KUKA KRL program: MyProgram_100().src

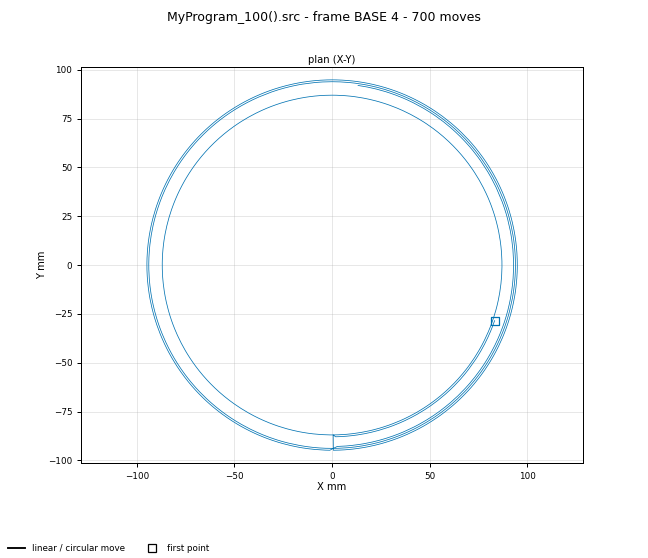
[picture p0: tool path of MyProgram_100().src in frame BASE 4, 700 of 700 moves have a stored position in this frame; points joined in program order, loops and branches not executed]
&ACCESS RVP
&REL 1
&PARAM TEMPLATE = C:\KRC\Roboter\Template\vorgabe
&PARAM EDITMASK = *
DEF MyProgram_100()
; ---- Setting reference (Base) ----
$BASE = BASE_DATA[4]

; --------------------------
; ---- Setting tool (TCP) ----
$TOOL = TOOL_DATA[3]
; --------------------------

$VEL.CP = VEL_APROX_PRINT
Startdeposition()
$VEL.CP = VEL_PRINT
LIN {X 83.2167,Y -28.4567,Z 91,A -24.2828,B 24.9207,C -2.0559,E1 25.1508,E2 469.2806} C_DIS
LIN {X 82.0556,Y -31.6498,Z 91,A -26.2319,B 24.9206,C -2.0583,E1 25.1489,E2 471.2131} C_DIS
LIN {X 81.1855,Y -33.8182,Z 91,A -28.5047,B 24.9229,C -2.0275,E1 25.1464,E2 473.5461} C_DIS
LIN {X 79.8483,Y -36.8641,Z 91,A -30.8218,B 24.9238,C -2.0158,E1 25.1436,E2 475.8782} C_DIS
LIN {X 78.1167,Y -40.407,Z 91,A -33.4521,B 24.9245,C -2.0061,E1 25.1403,E2 478.5174} C_DIS
LIN {X 76.1397,Y -44.0179,Z 91,A -35.2877,B 24.9229,C -2.0276,E1 25.1378,E2 480.2928} C_DIS
LIN {X 74.5815,Y -46.6088,Z 91,A -36.9718,B 24.9226,C -2.032,E1 25.1354,E2 481.958} C_DIS
LIN {X 73.464,Y -48.3511,Z 91,A -38.6448,B 24.9237,C -2.0169,E1 25.1328,E2 483.6583} C_DIS
LIN {X 69.7273,Y -53.5994,Z 91,A -42.6293,B 24.924,C -2.0128,E1 25.1263,E2 487.6331} C_DIS
LIN {X 67.7377,Y -56.0928,Z 91,A -44.8775,B 24.9249,C -2.0014,E1 25.1223,E2 489.8977} C_DIS
LIN {X 65.6016,Y -58.5766,Z 91,A -47.8573,B 24.9275,C -1.967,E1 25.1167,E2 492.9454} C_DIS
LIN {X 62.5852,Y -61.7889,Z 91,A -49.8249,B 24.9257,C -1.9908,E1 25.113,E2 494.8484} C_DIS
LIN {X 60.3828,Y -63.9431,Z 91,A -51.8518,B 24.9261,C -1.9854,E1 25.1089,E2 496.8799} C_DIS
LIN {X 57.9684,Y -66.1397,Z 91,A -54.9821,B 24.929,C -1.9464,E1 25.1022,E2 500.0897} C_DIS
LIN {X 54.1399,Y -69.31,Z 91,A -57.5673,B 24.9279,C -1.9614,E1 25.0966,E2 502.63} C_DIS
LIN {X 50.5294,Y -71.9838,Z 91,A -60.0241,B 24.9271,C -1.9713,E1 25.0911,E2 505.0547} C_DIS
LIN {X 47.6024,Y -73.9513,Z 91,A -62.3164,B 24.9275,C -1.967,E1 25.0858,E2 507.3495} C_DIS
LIN {X 43.6058,Y -76.3765,Z 91,A -65.9359,B 24.9293,C -1.9421,E1 25.0769,E2 511.0167} C_DIS
LIN {X 40.7609,Y -77.9317,Z 91,A -67.6031,B 24.9285,C -1.9534,E1 25.0729,E2 512.6526} C_DIS
LIN {X 37.3321,Y -79.6313,Z 91,A -69.9938,B 24.9285,C -1.9529,E1 25.0669,E2 515.0382} C_DIS
LIN {X 34.5175,Y -80.891,Z 91,A -72.0438,B 24.9288,C -1.9485,E1 25.0617,E2 517.0937} C_DIS
LIN {X 31.395,Y -82.1533,Z 91,A -73.9789,B 24.9284,C -1.9541,E1 25.0567,E2 519.0112} C_DIS
LIN {X 29.0169,Y -83.0229,Z 91,A -76.1026,B 24.9297,C -1.9362,E1 25.051,E2 521.1729} C_DIS
LIN {X 23.7913,Y -84.6686,Z 91,A -79.5291,B 24.9297,C -1.9368,E1 25.0419,E2 524.5919} C_DIS
LIN {X 20.0098,Y -85.6413,Z 91,A -82.0028,B 24.9297,C -1.9366,E1 25.0352,E2 527.0625} C_DIS
LIN {X 16.5913,Y -86.3684,Z 91,A -84.3026,B 24.9299,C -1.9339,E1 25.0288,E2 529.3658} C_DIS
LIN {X 13.0968,Y -86.9676,Z 91,A -86.358,B 24.9294,C -1.9405,E1 25.0232,E2 531.4036} C_DIS
LIN {X 10.7294,Y -87.291,Z 91,A -88.0802,B 24.9299,C -1.9341,E1 25.0184,E2 533.1395} C_DIS
LIN {X 7.6095,Y -87.6177,Z 91,A -90.1493,B 24.93,C -1.9322,E1 25.0127,E2 535.2119} C_DIS
LIN {X 4.3054,Y -87.8424,Z 91,A -92.3321,B 24.9301,C -1.9305,E1 25.0066,E2 537.3979} C_DIS
LIN {X 1.8163,Y -87.929,Z 91,A -93.8282,B 24.9299,C -1.934,E1 25.0024,E2 538.8854} C_DIS
LIN {X 1.8163,Y -87.929,Z 91,A -93.8282,B 24.9299,C -1.934,E1 25.0024,E2 538.8854} C_DIS
Enddeposition()
LIN {X 0.5508,Y -86.9757,Z 91,A -94.1889,B 24.9276,C -1.9656,E1 25.0016,E2 539.171} C_DIS
Startdeposition()
$VEL.CP = VEL_PRINT
LIN {X 3.2037,Y -86.9212,Z 91,A -92.2114,B 24.927,C -1.9735,E1 25.0072,E2 537.1751} C_DIS
LIN {X 5.3312,Y -86.8173,Z 91,A -90.8306,B 24.927,C -1.9734,E1 25.011,E2 535.7952} C_DIS
LIN {X 7.5293,Y -86.6532,Z 91,A -89.1451,B 24.9264,C -1.9817,E1 25.0158,E2 534.0908} C_DIS
LIN {X 10.6333,Y -86.3277,Z 91,A -87.3159,B 24.9268,C -1.9755,E1 25.0208,E2 532.2777} C_DIS
LIN {X 12.6686,Y -86.0529,Z 91,A -85.9635,B 24.9268,C -1.9764,E1 25.0246,E2 530.9243} C_DIS
LIN {X 14.7955,Y -85.7133,Z 91,A -84.5308,B 24.9266,C -1.9779,E1 25.0285,E2 529.4895} C_DIS
LIN {X 16.8911,Y -85.3246,Z 91,A -83.0893,B 24.9265,C -1.9803,E1 25.0325,E2 528.0439} C_DIS
LIN {X 19.0492,Y -84.8684,Z 91,A -81.6996,B 24.9265,C -1.9796,E1 25.0363,E2 526.6578} C_DIS
LIN {X 21.1564,Y -84.3677,Z 91,A -80.0242,B 24.9258,C -1.9892,E1 25.0409,E2 524.9621} C_DIS
LIN {X 24.1141,Y -83.57,Z 91,A -78.2555,B 24.9263,C -1.9832,E1 25.0456,E2 523.2107} C_DIS
LIN {X 26.0935,Y -82.9736,Z 91,A -76.8469,B 24.926,C -1.9863,E1 25.0493,E2 521.7972} C_DIS
LIN {X 28.8765,Y -82.0464,Z 91,A -74.8223,B 24.9256,C -1.9918,E1 25.0547,E2 519.7636} C_DIS
LIN {X 31.1689,Y -81.2034,Z 91,A -73.2999,B 24.9256,C -1.9911,E1 25.0587,E2 518.2461} C_DIS
LIN {X 33.2121,Y -80.389,Z 91,A -71.9115,B 24.9256,C -1.9911,E1 25.0623,E2 516.8608} C_DIS
LIN {X 35.1707,Y -79.5517,Z 91,A -70.5232,B 24.9256,C -1.9927,E1 25.0658,E2 515.472} C_DIS
LIN {X 37.1076,Y -78.6671,Z 91,A -68.9087,B 24.9248,C -2.002,E1 25.0699,E2 513.8396} C_DIS
LIN {X 39.9862,Y -77.2445,Z 91,A -66.7842,B 24.9246,C -2.0058,E1 25.0752,E2 511.712} C_DIS
LIN {X 42.7562,Y -75.7465,Z 91,A -64.9422,B 24.9249,C -2.0016,E1 25.0797,E2 509.8854} C_DIS
LIN {X 44.5558,Y -74.7018,Z 91,A -63.5773,B 24.9247,C -2.0039,E1 25.083,E2 508.5192} C_DIS
LIN {X 47.0289,Y -73.1693,Z 91,A -61.5921,B 24.9243,C -2.0099,E1 25.0877,E2 506.5262} C_DIS
LIN {X 48.8455,Y -71.9694,Z 91,A -60.1397,B 24.924,C -2.0133,E1 25.0911,E2 505.0705} C_DIS
LIN {X 50.8905,Y -70.539,Z 91,A -58.5953,B 24.924,C -2.0133,E1 25.0946,E2 503.5315} C_DIS
LIN {X 53.0933,Y -68.8953,Z 91,A -56.6917,B 24.9235,C -2.0203,E1 25.0988,E2 501.6182} C_DIS
LIN {X 55.5445,Y -66.9349,Z 91,A -54.6246,B 24.9231,C -2.0248,E1 25.1033,E2 499.5482} C_DIS
LIN {X 57.9872,Y -64.8302,Z 91,A -52.4847,B 24.9227,C -2.0302,E1 25.1078,E2 497.4041} C_DIS
LIN {X 60.3294,Y -62.6564,Z 91,A -50.4216,B 24.9224,C -2.0338,E1 25.112,E2 495.3411} C_DIS
LIN {X 62.6022,Y -60.3857,Z 91,A -48.3282,B 24.9221,C -2.0382,E1 25.1161,E2 493.2463} C_DIS
LIN {X 64.7171,Y -58.1135,Z 91,A -46.2361,B 24.9216,C -2.0449,E1 25.1201,E2 491.1474} C_DIS
LIN {X 66.8928,Y -55.5951,Z 91,A -44.092,B 24.9213,C -2.0489,E1 25.1239,E2 489.0036} C_DIS
LIN {X 68.8721,Y -53.1234,Z 91,A -42.0124,B 24.9209,C -2.0543,E1 25.1275,E2 486.9213} C_DIS
LIN {X 70.4344,Y -51.0353,Z 91,A -40.4263,B 24.9209,C -2.0543,E1 25.1301,E2 485.3426} C_DIS
LIN {X 71.6523,Y -49.311,Z 91,A -39.0478,B 24.9206,C -2.0578,E1 25.1323,E2 483.9628} C_DIS
LIN {X 72.9068,Y -47.4363,Z 91,A -37.6066,B 24.9204,C -2.0604,E1 25.1346,E2 482.5226} C_DIS
LIN {X 74.0526,Y -45.6272,Z 91,A -36.1871,B 24.9201,C -2.0647,E1 25.1367,E2 481.1002} C_DIS
LIN {X 75.1471,Y -43.8021,Z 91,A -34.6258,B 24.9193,C -2.0743,E1 25.1389,E2 479.5242} C_DIS
LIN {X 76.6816,Y -41.0553,Z 91,A -32.7076,B 24.9193,C -2.0749,E1 25.1415,E2 477.6144} C_DIS
LIN {X 77.9149,Y -38.6618,Z 91,A -30.7952,B 24.9185,C -2.085,E1 25.1439,E2 475.6884} C_DIS
LIN {X 79.0625,Y -36.2567,Z 91,A -29.2221,B 24.9185,C -2.0839,E1 25.1457,E2 474.1264} C_DIS
LIN {X 79.915,Y -34.3382,Z 91,A -27.8263,B 24.9182,C -2.0885,E1 25.1473,E2 472.7273} C_DIS
LIN {X 81.0139,Y -31.6582,Z 91,A -25.823,B 24.9175,C -2.0977,E1 25.1494,E2 470.7135} C_DIS
LIN {X 81.8944,Y -29.306,Z 91,A -24.3434,B 24.9175,C -2.0967,E1 25.1508,E2 469.2445} C_DIS
LIN {X 82.564,Y -27.3612,Z 91,A -22.9651,B 24.9172,C -2.1017,E1 25.152,E2 467.8621} C_DIS
LIN {X 83.2312,Y -25.2607,Z 91,A -21.5144,B 24.9168,C -2.1062,E1 25.1532,E2 466.4091} C_DIS
LIN {X 83.8304,Y -23.1943,Z 91,A -20.1436,B 24.9166,C -2.109,E1 25.1543,E2 465.0394} C_DIS
LIN {X 84.4419,Y -20.8587,Z 91,A -18.3066,B 24.9155,C -2.1227,E1 25.1555,E2 463.1807} C_DIS
LIN {X 85.0643,Y -18.1527,Z 91,A -16.7409,B 24.9158,C -2.1193,E1 25.1565,E2 461.6323} C_DIS
LIN {X 85.4869,Y -16.0474,Z 91,A -15.3263,B 24.9154,C -2.1238,E1 25.1572,E2 460.2153} C_DIS
LIN {X 85.8311,Y -14.0906,Z 91,A -13.9881,B 24.915,C -2.129,E1 25.1579,E2 458.8727} C_DIS
LIN {X 86.1885,Y -11.7095,Z 91,A -12.4573,B 24.9147,C -2.1321,E1 25.1585,E2 457.3435} C_DIS
LIN {X 86.4429,Y -9.6511,Z 91,A -11.0636,B 24.9143,C -2.1375,E1 25.1589,E2 455.9454} C_DIS
LIN {X 86.653,Y -7.5314,Z 91,A -9.7473,B 24.9142,C -2.139,E1 25.1593,E2 454.6334} C_DIS
LIN {X 86.8123,Y -5.4068,Z 91,A -8.2791,B 24.9136,C -2.1457,E1 25.1595,E2 453.158} C_DIS
LIN {X 86.9211,Y -3.2052,Z 91,A -6.8454,B 24.9133,C -2.1497,E1 25.1597,E2 451.7233} C_DIS
LIN {X 86.9756,Y -0.9547,Z 91,A -5.1249,B 24.9123,C -2.1628,E1 25.1597,E2 449.9821} C_DIS
LIN {X 86.9553,Y 2.0675,Z 91,A -3.3966,B 24.9125,C -2.16,E1 25.1597,E2 448.2709} C_DIS
LIN {X 86.8784,Y 4.1974,Z 91,A -2.0346,B 24.9122,C -2.163,E1 25.1595,E2 446.9098} C_DIS
LIN {X 86.7456,Y 6.3985,Z 91,A -0.2652,B 24.911,C -2.1787,E1 25.1592,E2 445.1138} C_DIS
LIN {X 86.4587,Y 9.5085,Z 91,A 1.6567,B 24.9108,C -2.1805,E1 25.1586,E2 443.1991} C_DIS
LIN {X 86.0492,Y 12.6942,Z 91,A 3.568,B 24.9108,C -2.18,E1 25.1579,E2 441.3003} C_DIS
LIN {X 85.7127,Y 14.7989,Z 91,A 4.9825,B 24.9105,C -2.1847,E1 25.1573,E2 439.883} C_DIS
LIN {X 85.3239,Y 16.8945,Z 91,A 6.4155,B 24.91,C -2.1901,E1 25.1565,E2 438.4456} C_DIS
LIN {X 84.8193,Y 19.2669,Z 91,A 8.1959,B 24.9091,C -2.2014,E1 25.1554,E2 436.6488} C_DIS
LIN {X 84.1069,Y 22.1706,Z 91,A 9.9085,B 24.9093,C -2.1985,E1 25.1543,E2 434.9531} C_DIS
LIN {X 83.3271,Y 24.9422,Z 91,A 11.8642,B 24.9087,C -2.2062,E1 25.1527,E2 432.9902} C_DIS
LIN {X 82.624,Y 27.1791,Z 91,A 13.4914,B 24.9081,C -2.2137,E1 25.1513,E2 431.3545} C_DIS
LIN {X 81.5552,Y 30.2355,Z 91,A 15.4262,B 24.9081,C -2.2131,E1 25.1495,E2 429.432} C_DIS
LIN {X 80.8419,Y 32.0944,Z 91,A 16.802,B 24.9076,C -2.2192,E1 25.1481,E2 428.0496} C_DIS
LIN {X 79.9497,Y 34.2571,Z 91,A 18.2728,B 24.9075,C -2.2211,E1 25.1465,E2 426.5821} C_DIS
LIN {X 78.9634,Y 36.4723,Z 91,A 20.0777,B 24.9065,C -2.2329,E1 25.1444,E2 424.7595} C_DIS
LIN {X 77.4059,Y 39.6711,Z 91,A 22.3006,B 24.9063,C -2.2352,E1 25.1417,E2 422.5429} C_DIS
LIN {X 76.1964,Y 41.9495,Z 91,A 23.857,B 24.9063,C -2.2349,E1 25.1396,E2 420.9954} C_DIS
LIN {X 75.2363,Y 43.6472,Z 91,A 25.1847,B 24.9059,C -2.2398,E1 25.1378,E2 419.663} C_DIS
LIN {X 74.0934,Y 45.5609,Z 91,A 26.6123,B 24.9057,C -2.2422,E1 25.1357,E2 418.2368} C_DIS
LIN {X 72.9171,Y 47.4205,Z 91,A 28.0297,B 24.9055,C -2.2449,E1 25.1336,E2 416.8203} C_DIS
LIN {X 71.7788,Y 49.1265,Z 91,A 29.5574,B 24.9047,C -2.2544,E1 25.1311,E2 415.2777} C_DIS
LIN {X 69.8641,Y 51.8135,Z 91,A 31.5363,B 24.9047,C -2.2531,E1 25.1279,E2 413.3115} C_DIS
LIN {X 68.2433,Y 53.9289,Z 91,A 33.4574,B 24.9039,C -2.263,E1 25.1246,E2 411.3761} C_DIS
LIN {X 66.2325,Y 56.3801,Z 91,A 35.528,B 24.9036,C -2.2672,E1 25.1209,E2 409.3049} C_DIS
LIN {X 64.0975,Y 58.7961,Z 91,A 37.6276,B 24.9032,C -2.2712,E1 25.117,E2 407.2053} C_DIS
LIN {X 61.9023,Y 61.103,Z 91,A 39.6528,B 24.9031,C -2.2732,E1 25.113,E2 405.184} C_DIS
LIN {X 59.6715,Y 63.2834,Z 91,A 41.8334,B 24.9023,C -2.2817,E1 25.1086,E2 402.9923} C_DIS
LIN {X 56.806,Y 65.8694,Z 91,A 44.381,B 24.9019,C -2.2869,E1 25.1033,E2 400.4426} C_DIS
LIN {X 54.3557,Y 67.9053,Z 91,A 46.4557,B 24.9016,C -2.29,E1 25.0988,E2 398.3685} C_DIS
LIN {X 51.8327,Y 69.8498,Z 91,A 48.3364,B 24.9019,C -2.2865,E1 25.0946,E2 396.5029} C_DIS
LIN {X 50.1143,Y 71.0928,Z 91,A 49.7213,B 24.9017,C -2.2884,E1 25.0915,E2 395.1183} C_DIS
LIN {X 48.3276,Y 72.32,Z 91,A 51.2092,B 24.9014,C -2.2927,E1 25.088,E2 393.6251} C_DIS
LIN {X 46.6021,Y 73.443,Z 91,A 52.7575,B 24.9006,C -2.3012,E1 25.0844,E2 392.0617} C_DIS
LIN {X 43.7946,Y 75.1514,Z 91,A 54.6744,B 24.9011,C -2.2962,E1 25.0798,E2 390.1627} C_DIS
LIN {X 42.1288,Y 76.0968,Z 91,A 55.9691,B 24.9008,C -2.299,E1 25.0767,E2 388.865} C_DIS
LIN {X 40.1328,Y 77.1678,Z 91,A 57.3992,B 24.9008,C -2.299,E1 25.0731,E2 387.4391} C_DIS
LIN {X 38.2334,Y 78.1259,Z 91,A 58.8479,B 24.9006,C -2.3023,E1 25.0695,E2 385.9864} C_DIS
LIN {X 36.2219,Y 79.0785,Z 91,A 60.4307,B 24.9001,C -2.3078,E1 25.0655,E2 384.3945} C_DIS
LIN {X 33.3591,Y 80.328,Z 91,A 62.3607,B 24.9002,C -2.3059,E1 25.0605,E2 382.4738} C_DIS
LIN {X 31.3818,Y 81.1218,Z 91,A 63.6826,B 24.9004,C -2.3046,E1 25.0571,E2 381.1578} C_DIS
LIN {X 29.3004,Y 81.8964,Z 91,A 65.1628,B 24.9002,C -2.3065,E1 25.0532,E2 379.6762} C_DIS
LIN {X 26.8533,Y 82.7307,Z 91,A 67.0718,B 24.8995,C -2.3146,E1 25.0481,E2 377.7517} C_DIS
LIN {X 24.308,Y 83.5139,Z 91,A 68.6499,B 24.8999,C -2.3102,E1 25.0439,E2 376.1869} C_DIS
LIN {X 22.2486,Y 84.0865,Z 91,A 70.2341,B 24.8993,C -2.3167,E1 25.0396,E2 374.5896} C_DIS
LIN {X 19.099,Y 84.8571,Z 91,A 72.3825,B 24.8992,C -2.3183,E1 25.0338,E2 372.4406} C_DIS
LIN {X 15.918,Y 85.5115,Z 91,A 74.3105,B 24.8997,C -2.3124,E1 25.0286,E2 370.5288} C_DIS
LIN {X 13.8178,Y 85.8767,Z 91,A 75.7258,B 24.8997,C -2.3132,E1 25.0247,E2 369.113} C_DIS
LIN {X 11.7091,Y 86.1886,Z 91,A 77.1129,B 24.8997,C -2.3131,E1 25.0208,E2 367.7275} C_DIS
LIN {X 9.6669,Y 86.4412,Z 91,A 78.5079,B 24.8995,C -2.3146,E1 25.0169,E2 366.3299} C_DIS
LIN {X 6.6709,Y 86.7238,Z 91,A 80.5114,B 24.8995,C -2.3154,E1 25.0114,E2 364.3256} C_DIS
LIN {X 4.3419,Y 86.8717,Z 91,A 82.0277,B 24.8995,C -2.3147,E1 25.0072,E2 362.8115} C_DIS
LIN {X 2.2117,Y 86.9515,Z 91,A 83.4025,B 24.8995,C -2.3137,E1 25.0033,E2 361.4395} C_DIS
LIN {X 0.0073,Y 86.9813,Z 91,A 85.1448,B 24.8988,C -2.3225,E1 24.9984,E2 359.6764} C_DIS
LIN {X -3.6285,Y 86.904,Z 91,A 87.4261,B 24.8992,C -2.3182,E1 24.9921,E2 357.4049} C_DIS
LIN {X -6.3998,Y 86.7454,Z 91,A 89.1398,B 24.8995,C -2.3139,E1 24.9873,E2 355.7009} C_DIS
LIN {X -8.8241,Y 86.5312,Z 91,A 90.9283,B 24.8991,C -2.3188,E1 24.9823,E2 353.8996} C_DIS
LIN {X -11.6977,Y 86.1901,Z 91,A 92.5734,B 24.8999,C -2.3096,E1 24.9778,E2 352.2752} C_DIS
LIN {X -13.8043,Y 85.8788,Z 91,A 94.1856,B 24.8994,C -2.3151,E1 24.9733,E2 350.6485} C_DIS
LIN {X -16.8956,Y 85.3237,Z 91,A 96.1315,B 24.8999,C -2.3097,E1 24.968,E2 348.7134} C_DIS
LIN {X -19.0504,Y 84.8681,Z 91,A 97.537,B 24.9001,C -2.3071,E1 24.9642,E2 347.3124} C_DIS
LIN {X -21.0786,Y 84.3872,Z 91,A 98.9317,B 24.9001,C -2.3064,E1 24.9604,E2 345.9173} C_DIS
LIN {X -23.2048,Y 83.8275,Z 91,A 100.566,B 24.8998,C -2.3106,E1 24.956,E2 344.2706} C_DIS
LIN {X -26.1917,Y 82.9428,Z 91,A 102.444,B 24.9005,C -2.303,E1 24.951,E2 342.4074} C_DIS
LIN {X -28.8203,Y 82.0662,Z 91,A 104.3862,B 24.9004,C -2.3043,E1 24.9458,E2 340.4584} C_DIS
LIN {X -31.204,Y 81.1899,Z 91,A 105.9711,B 24.9008,C -2.2995,E1 24.9417,E2 338.8817} C_DIS
LIN {X -33.6895,Y 80.1903,Z 91,A 107.8745,B 24.9006,C -2.3012,E1 24.9368,E2 336.9699} C_DIS
LIN {X -36.1488,Y 79.1121,Z 91,A 109.6649,B 24.9008,C -2.2992,E1 24.9322,E2 335.1799} C_DIS
LIN {X -39.1143,Y 77.6889,Z 91,A 111.5954,B 24.9017,C -2.2887,E1 24.9274,E2 333.2693} C_DIS
LIN {X -41.0039,Y 76.7092,Z 91,A 113.0442,B 24.9018,C -2.2878,E1 24.9238,E2 331.8188} C_DIS
LIN {X -42.8037,Y 75.72,Z 91,A 114.4231,B 24.9019,C -2.2862,E1 24.9205,E2 330.4397} C_DIS
LIN {X -44.6426,Y 74.6502,Z 91,A 115.8187,B 24.9022,C -2.2835,E1 24.9171,E2 329.0462} C_DIS
LIN {X -46.4539,Y 73.537,Z 91,A 117.2624,B 24.9022,C -2.2822,E1 24.9137,E2 327.6011} C_DIS
LIN {X -48.2366,Y 72.3801,Z 91,A 118.6449,B 24.9026,C -2.279,E1 24.9105,E2 326.2217} C_DIS
LIN {X -50.3981,Y 70.8909,Z 91,A 120.5441,B 24.9024,C -2.2806,E1 24.9061,E2 324.3123} C_DIS
LIN {X -53.0437,Y 68.9336,Z 91,A 122.6632,B 24.9029,C -2.2746,E1 24.9014,E2 322.1997} C_DIS
LIN {X -55.4221,Y 67.0366,Z 91,A 124.7441,B 24.9031,C -2.2725,E1 24.8969,E2 320.116} C_DIS
LIN {X -58.0076,Y 64.8119,Z 91,A 126.9209,B 24.9037,C -2.2654,E1 24.8923,E2 317.9475} C_DIS
LIN {X -60.3403,Y 62.6459,Z 91,A 129.0435,B 24.9041,C -2.2613,E1 24.888,E2 315.8261} C_DIS
LIN {X -62.6248,Y 60.3622,Z 91,A 131.1927,B 24.9045,C -2.2567,E1 24.8838,E2 313.6785} C_DIS
LIN {X -64.7984,Y 58.0227,Z 91,A 133.265,B 24.905,C -2.2506,E1 24.8799,E2 311.6118} C_DIS
LIN {X -66.9013,Y 55.5849,Z 91,A 135.4229,B 24.9053,C -2.2462,E1 24.876,E2 309.4544} C_DIS
LIN {X -68.9049,Y 53.0809,Z 91,A 137.5808,B 24.9057,C -2.242,E1 24.8723,E2 307.2965} C_DIS
LIN {X -70.467,Y 50.9902,Z 91,A 139.1871,B 24.9064,C -2.2341,E1 24.8697,E2 305.7013} C_DIS
LIN {X -71.6878,Y 49.2599,Z 91,A 140.5789,B 24.9067,C -2.2302,E1 24.8675,E2 304.3119} C_DIS
LIN {X -73.2012,Y 46.9793,Z 91,A 142.5101,B 24.9068,C -2.2288,E1 24.8645,E2 302.3742} C_DIS
LIN {X -74.5887,Y 44.746,Z 91,A 144.1198,B 24.9075,C -2.2204,E1 24.8622,E2 300.7763} C_DIS
LIN {X -75.6527,Y 42.9225,Z 91,A 145.5412,B 24.9078,C -2.2173,E1 24.8602,E2 299.3549} C_DIS
LIN {X -77.0097,Y 40.4349,Z 91,A 147.5352,B 24.9079,C -2.2155,E1 24.8576,E2 297.3547} C_DIS
LIN {X -78.1325,Y 38.2199,Z 91,A 149.0767,B 24.9085,C -2.208,E1 24.8557,E2 295.8227} C_DIS
LIN {X -79.0758,Y 36.2279,Z 91,A 150.5194,B 24.9089,C -2.2034,E1 24.854,E2 294.3832} C_DIS
LIN {X -80.148,Y 33.7899,Z 91,A 152.4546,B 24.9089,C -2.2033,E1 24.8518,E2 292.4377} C_DIS
LIN {X -81.1252,Y 31.3729,Z 91,A 154.1733,B 24.9094,C -2.198,E1 24.8501,E2 290.7218} C_DIS
LIN {X -82.2299,Y 28.3515,Z 91,A 156.1809,B 24.9102,C -2.1884,E1 24.8482,E2 288.7259} C_DIS
LIN {X -82.9211,Y 26.2607,Z 91,A 157.6074,B 24.9106,C -2.1832,E1 24.847,E2 287.3036} C_DIS
LIN {X -83.5181,Y 24.2934,Z 91,A 158.9715,B 24.9109,C -2.1792,E1 24.8459,E2 285.941} C_DIS
LIN {X -84.0883,Y 22.2415,Z 91,A 160.386,B 24.9113,C -2.1752,E1 24.8449,E2 284.528} C_DIS
LIN {X -84.6244,Y 20.1038,Z 91,A 161.8272,B 24.9117,C -2.1703,E1 24.8439,E2 283.09} C_DIS
LIN {X -85.0758,Y 18.0987,Z 91,A 163.1914,B 24.912,C -2.1663,E1 24.8431,E2 281.7273} C_DIS
LIN {X -85.5074,Y 15.9394,Z 91,A 164.8569,B 24.9119,C -2.1678,E1 24.8422,E2 280.0485} C_DIS
LIN {X -86.0263,Y 12.8507,Z 91,A 166.7847,B 24.9127,C -2.1573,E1 24.8414,E2 278.1341} C_DIS
LIN {X -86.3119,Y 10.7628,Z 91,A 168.1558,B 24.9131,C -2.1524,E1 24.8409,E2 276.7665} C_DIS
LIN {X -86.5922,Y 8.2037,Z 91,A 170.0421,B 24.9131,C -2.1524,E1 24.8404,E2 274.8689} C_DIS
LIN {X -86.81,Y 5.4415,Z 91,A 171.6855,B 24.914,C -2.1414,E1 24.84,E2 273.2419} C_DIS
LIN {X -86.9189,Y 3.2716,Z 91,A 173.1701,B 24.9142,C -2.1383,E1 24.8399,E2 271.7558} C_DIS
LIN {X -86.9756,Y 0.9538,Z 91,A 174.9257,B 24.9142,C -2.1399,E1 24.8398,E2 269.9857} C_DIS
LIN {X -86.9564,Y -2.0256,Z 91,A 176.6613,B 24.9151,C -2.1272,E1 24.8398,E2 268.27} C_DIS
LIN {X -86.8814,Y -4.1347,Z 91,A 178.0082,B 24.9156,C -2.1216,E1 24.84,E2 266.9285} C_DIS
LIN {X -86.7522,Y -6.3022,Z 91,A 179.7612,B 24.9152,C -2.1262,E1 24.8404,E2 265.154} C_DIS
LIN {X -86.4611,Y -9.4869,Z 91,A -178.3728,B 24.9163,C -2.1127,E1 24.8409,E2 263.309} C_DIS
LIN {X -86.1984,Y -11.6349,Z 91,A -176.992,B 24.9167,C -2.1069,E1 24.8414,E2 261.9336} C_DIS
LIN {X -85.9008,Y -13.6624,Z 91,A -175.6092,B 24.917,C -2.1036,E1 24.8419,E2 260.5505} C_DIS
LIN {X -85.4637,Y -16.1692,Z 91,A -173.7453,B 24.917,C -2.1038,E1 24.8429,E2 258.6752} C_DIS
LIN {X -84.8889,Y -18.9583,Z 91,A -172,B 24.9177,C -2.0943,E1 24.8439,E2 256.9422} C_DIS
LIN {X -84.3979,Y -21.0356,Z 91,A -170.5826,B 24.9181,C -2.0903,E1 24.8448,E2 255.526} C_DIS
LIN {X -83.8423,Y -23.1513,Z 91,A -169.1391,B 24.9184,C -2.086,E1 24.8459,E2 254.0844} C_DIS
LIN {X -83.0872,Y -25.7291,Z 91,A -167.2117,B 24.9184,C -2.0852,E1 24.8474,E2 252.1477} C_DIS
LIN {X -82.249,Y -28.2955,Z 91,A -165.58,B 24.9192,C -2.0758,E1 24.8489,E2 250.5294} C_DIS
LIN {X -81.5561,Y -30.2329,Z 91,A -164.2384,B 24.9195,C -2.0714,E1 24.8502,E2 249.1906} C_DIS
LIN {X -80.547,Y -32.8274,Z 91,A -162.2249,B 24.9195,C -2.0713,E1 24.8522,E2 247.1662} C_DIS
LIN {X -79.215,Y -35.9234,Z 91,A -160.0508,B 24.9201,C -2.0636,E1 24.8547,E2 244.9983} C_DIS
LIN {X -78.1998,Y -38.083,Z 91,A -158.5328,B 24.9206,C -2.0577,E1 24.8565,E2 243.4862} C_DIS
LIN {X -77.2496,Y -39.9764,Z 91,A -157.1367,B 24.9209,C -2.0539,E1 24.8583,E2 242.0918} C_DIS
LIN {X -76.2009,Y -41.9414,Z 91,A -155.7028,B 24.9213,C -2.0489,E1 24.8602,E2 240.6621} C_DIS
LIN {X -75.1881,Y -43.731,Z 91,A -154.3072,B 24.9215,C -2.0465,E1 24.8621,E2 239.265} C_DIS
LIN {X -74.0946,Y -45.5589,Z 91,A -152.9122,B 24.9218,C -2.0426,E1 24.8641,E2 237.8721} C_DIS
LIN {X -72.6728,Y -47.7927,Z 91,A -151.0008,B 24.9218,C -2.043,E1 24.8671,E2 235.9502} C_DIS
LIN {X -71.1438,Y -50.0415,Z 91,A -149.3465,B 24.9224,C -2.0345,E1 24.8697,E2 234.308} C_DIS
LIN {X -69.8579,Y -51.8219,Z 91,A -147.9307,B 24.9227,C -2.0301,E1 24.872,E2 232.8959} C_DIS
LIN {X -68.2393,Y -53.9338,Z 91,A -145.9946,B 24.9227,C -2.0313,E1 24.8753,E2 230.9477} C_DIS
LIN {X -66.237,Y -56.3749,Z 91,A -143.9053,B 24.923,C -2.0267,E1 24.8791,E2 228.8596} C_DIS
LIN {X -64.0567,Y -58.8405,Z 91,A -141.8715,B 24.9236,C -2.0179,E1 24.8829,E2 226.8377} C_DIS
LIN {X -62.2845,Y -60.7151,Z 91,A -139.9372,B 24.9234,C -2.0212,E1 24.8866,E2 224.8872} C_DIS
LIN {X -59.995,Y -62.9777,Z 91,A -137.8467,B 24.9238,C -2.016,E1 24.8908,E2 222.8006} C_DIS
LIN {X -57.6171,Y -65.1609,Z 91,A -135.6927,B 24.9241,C -2.0126,E1 24.8953,E2 220.646} C_DIS
LIN {X -55.1871,Y -67.2309,Z 91,A -133.581,B 24.9243,C -2.0089,E1 24.8998,E2 218.535} C_DIS
LIN {X -52.7136,Y -69.1875,Z 91,A -131.539,B 24.9247,C -2.0041,E1 24.9043,E2 216.4969} C_DIS
LIN {X -50.0868,Y -71.1121,Z 91,A -129.5748,B 24.9254,C -1.9951,E1 24.9087,E2 214.5474} C_DIS
LIN {X -48.4103,Y -72.264,Z 91,A -128.146,B 24.9254,C -1.9956,E1 24.912,E2 213.1126} C_DIS
LIN {X -46.5932,Y -73.4486,Z 91,A -126.7369,B 24.9255,C -1.9928,E1 24.9153,E2 211.7056} C_DIS
LIN {X -44.719,Y -74.6048,Z 91,A -125.3175,B 24.9258,C -1.9897,E1 24.9187,E2 210.2892} C_DIS
LIN {X -42.8806,Y -75.6767,Z 91,A -123.6699,B 24.9254,C -1.9953,E1 24.9228,E2 208.6235} C_DIS
LIN {X -40.1237,Y -77.1726,Z 91,A -121.795,B 24.926,C -1.9867,E1 24.9274,E2 206.7636} C_DIS
LIN {X -37.5444,Y -78.4595,Z 91,A -119.7917,B 24.926,C -1.9877,E1 24.9324,E2 204.7529} C_DIS
LIN {X -35.2534,Y -79.515,Z 91,A -118.0595,B 24.9259,C -1.988,E1 24.9368,E2 203.0157} C_DIS
LIN {X -32.2945,Y -80.7619,Z 91,A -116.196,B 24.9266,C -1.9781,E1 24.9416,E2 201.1715} C_DIS
LIN {X -29.8277,Y -81.7054,Z 91,A -114.2664,B 24.9263,C -1.9824,E1 24.9467,E2 199.2277} C_DIS
LIN {X -27.3647,Y -82.5628,Z 91,A -112.6726,B 24.9267,C -1.9772,E1 24.9509,E2 197.6433} C_DIS
LIN {X -25.2584,Y -83.2319,Z 91,A -111.208,B 24.9267,C -1.9764,E1 24.9548,E2 196.1781} C_DIS
LIN {X -23.2314,Y -83.8202,Z 91,A -109.5935,B 24.9263,C -1.9825,E1 24.9591,E2 194.5465} C_DIS
LIN {X -19.8668,Y -84.6809,Z 91,A -107.2804,B 24.9263,C -1.982,E1 24.9654,E2 192.2312} C_DIS
LIN {X -17.041,Y -85.2944,Z 91,A -105.6165,B 24.927,C -1.9736,E1 24.9699,E2 190.5854} C_DIS
LIN {X -14.8733,Y -85.6996,Z 91,A -104.1922,B 24.927,C -1.9722,E1 24.9738,E2 189.1629} C_DIS
LIN {X -12.2895,Y -86.1071,Z 91,A -102.3082,B 24.9267,C -1.9769,E1 24.9791,E2 187.2662} C_DIS
LIN {X -9.6719,Y -86.4406,Z 91,A -100.6806,B 24.927,C -1.9731,E1 24.9836,E2 185.6465} C_DIS
LIN {X -7.5359,Y -86.6526,Z 91,A -99.3407,B 24.9272,C -1.9707,E1 24.9873,E2 184.3117} C_DIS
LIN {X -5.4108,Y -86.812,Z 91,A -97.8727,B 24.927,C -1.9727,E1 24.9914,E2 182.8382} C_DIS
LIN {X -3.2083,Y -86.921,Z 91,A -96.4265,B 24.927,C -1.9727,E1 24.9954,E2 181.3919} C_DIS
LIN {X -1.078,Y -86.9736,Z 91,A -95.0797,B 24.9272,C -1.9711,E1 24.9992,E2 180.0488} C_DIS
LIN {X 0.5508,Y -86.9757,Z 91,A -94.1887,B 24.9276,C -1.9655,E1 25.0016,E2 179.171} C_DIS
Enddeposition()
LIN {X 0.6401,Y -94.826,Z 92,A -93.7106,B 24.9358,C -1.8511,E1 25.0022,E2 178.9645} C_DIS
Startdeposition()
$VEL.CP = VEL_PRINT
LIN {X 3.7727,Y -94.7555,Z 92,A -91.7074,B 24.9355,C -1.8556,E1 25.0078,E2 176.9511} C_DIS
LIN {X 6.6945,Y -94.594,Z 92,A -89.8345,B 24.9351,C -1.8601,E1 25.0131,E2 175.0683} C_DIS
LIN {X 10.4526,Y -94.2541,Z 92,A -87.5882,B 24.9351,C -1.8601,E1 25.0193,E2 172.8233} C_DIS
LIN {X 13.0422,Y -93.9294,Z 92,A -86.0454,B 24.9351,C -1.8599,E1 25.0236,E2 171.2822} C_DIS
LIN {X 16.2126,Y -93.4357,Z 92,A -84.2042,B 24.9353,C -1.8578,E1 25.0286,E2 169.4478} C_DIS
LIN {X 18.5008,Y -93.0097,Z 92,A -82.6739,B 24.9349,C -1.8635,E1 25.0328,E2 167.9059} C_DIS
LIN {X 21.9117,Y -92.2657,Z 92,A -80.5691,B 24.9348,C -1.8653,E1 25.0386,E2 165.7997} C_DIS
LIN {X 25.2929,Y -91.3967,Z 92,A -78.4645,B 24.9346,C -1.8674,E1 25.0443,E2 163.6936} C_DIS
LIN {X 27.5282,Y -90.7485,Z 92,A -77.0257,B 24.9344,C -1.8702,E1 25.0481,E2 162.2506} C_DIS
LIN {X 30.8498,Y -89.6737,Z 92,A -75.0844,B 24.9347,C -1.8666,E1 25.0532,E2 160.3215} C_DIS
LIN {X 33.3053,Y -88.7896,Z 92,A -73.5123,B 24.9346,C -1.8686,E1 25.0574,E2 158.748} C_DIS
LIN {X 35.7443,Y -87.8356,Z 92,A -71.8245,B 24.9341,C -1.8747,E1 25.0618,E2 157.0496} C_DIS
LIN {X 38.6873,Y -86.5802,Z 92,A -70.1646,B 24.9346,C -1.8675,E1 25.066,E2 155.4107} C_DIS
LIN {X 40.8004,Y -85.6047,Z 92,A -68.7633,B 24.9345,C -1.8695,E1 25.0695,E2 154.0082} C_DIS
LIN {X 42.6375,Y -84.7061,Z 92,A -67.2489,B 24.9336,C -1.8818,E1 25.0734,E2 152.4688} C_DIS
LIN {X 44.7034,Y -83.6343,Z 92,A -65.8477,B 24.9335,C -1.884,E1 25.0768,E2 151.0664} C_DIS
LIN {X 46.7425,Y -82.512,Z 92,A -64.447,B 24.9333,C -1.8863,E1 25.0802,E2 149.6643} C_DIS
LIN {X 48.7533,Y -81.34,Z 92,A -63.0464,B 24.9331,C -1.8887,E1 25.0836,E2 148.2625} C_DIS
LIN {X 51.2383,Y -79.7959,Z 92,A -61.3096,B 24.933,C -1.8909,E1 25.0877,E2 146.5259} C_DIS
LIN {X 53.8813,Y -78.0361,Z 92,A -59.6584,B 24.9334,C -1.8848,E1 25.0915,E2 144.8949} C_DIS
LIN {X 55.7802,Y -76.6903,Z 92,A -58.102,B 24.9328,C -1.8933,E1 25.095,E2 143.3238} C_DIS
LIN {X 58.5652,Y -74.5853,Z 92,A -56.1591,B 24.9329,C -1.8915,E1 25.0993,E2 141.3921} C_DIS
LIN {X 60.1607,Y -73.306,Z 92,A -54.6467,B 24.932,C -1.9046,E1 25.1027,E2 139.8545} C_DIS
LIN {X 61.9416,Y -71.8075,Z 92,A -53.2474,B 24.9318,C -1.9075,E1 25.1056,E2 138.4537} C_DIS
LIN {X 63.8933,Y -70.0748,Z 92,A -51.8044,B 24.9318,C -1.9062,E1 25.1086,E2 137.0197} C_DIS
LIN {X 65.5938,Y -68.4857,Z 92,A -50.4055,B 24.9317,C -1.9092,E1 25.1114,E2 135.6194} C_DIS
LIN {X 67.8952,Y -66.2065,Z 92,A -48.4755,B 24.9314,C -1.913,E1 25.1153,E2 133.6888} C_DIS
LIN {X 69.5512,Y -64.464,Z 92,A -47.0734,B 24.9313,C -1.9147,E1 25.1179,E2 132.2887} C_DIS
LIN {X 71.2278,Y -62.6054,Z 92,A -45.6668,B 24.9313,C -1.9145,E1 25.1205,E2 130.8887} C_DIS
LIN {X 72.7428,Y -60.8385,Z 92,A -44.1119,B 24.9306,C -1.9238,E1 25.1234,E2 129.319} C_DIS
LIN {X 74.9328,Y -58.1198,Z 92,A -42.1713,B 24.9306,C -1.923,E1 25.1267,E2 127.3893} C_DIS
LIN {X 76.4997,Y -56.0406,Z 92,A -40.3363,B 24.9296,C -1.9373,E1 25.1298,E2 125.5295} C_DIS
LIN {X 78.1974,Y -53.6494,Z 92,A -38.5639,B 24.9293,C -1.9421,E1 25.1327,E2 123.7542} C_DIS
LIN {X 80.1191,Y -50.7348,Z 92,A -36.4673,B 24.9289,C -1.9476,E1 25.1358,E2 121.6553} C_DIS
LIN {X 81.34,Y -48.7533,Z 92,A -35.0699,B 24.9286,C -1.9513,E1 25.1379,E2 120.2563} C_DIS
LIN {X 82.512,Y -46.7425,Z 92,A -33.6726,B 24.9283,C -1.955,E1 25.1398,E2 118.8574} C_DIS
LIN {X 83.7078,Y -44.5637,Z 92,A -32.2526,B 24.9283,C -1.9563,E1 25.1417,E2 117.4418} C_DIS
LIN {X 85.223,Y -41.5948,Z 92,A -30.1795,B 24.9276,C -1.9646,E1 25.1443,E2 115.3603} C_DIS
LIN {X 86.301,Y -39.3068,Z 92,A -28.8991,B 24.928,C -1.9597,E1 25.1458,E2 114.0983} C_DIS
LIN {X 87.1613,Y -37.363,Z 92,A -27.5113,B 24.9274,C -1.9675,E1 25.1473,E2 112.6996} C_DIS
LIN {X 88.052,Y -35.2127,Z 92,A -26.1145,B 24.9271,C -1.9715,E1 25.1488,E2 111.3012} C_DIS
LIN {X 89.04,Y -32.629,Z 92,A -24.5167,B 24.927,C -1.9738,E1 25.1504,E2 109.7067} C_DIS
LIN {X 90.0456,Y -29.747,Z 92,A -22.4968,B 24.926,C -1.9863,E1 25.1522,E2 107.6688} C_DIS
LIN {X 90.7485,Y -27.5282,Z 92,A -21.1,B 24.9257,C -1.9903,E1 25.1533,E2 106.2705} C_DIS
LIN {X 91.3967,Y -25.2929,Z 92,A -19.6326,B 24.9252,C -1.9971,E1 25.1544,E2 104.7955} C_DIS
LIN {X 92.2657,Y -21.9117,Z 92,A -17.7343,B 24.9253,C -1.9957,E1 25.1557,E2 102.9115} C_DIS
LIN {X 92.8325,Y -19.3641,Z 92,A -16.1448,B 24.9249,C -2.0012,E1 25.1567,E2 101.3182} C_DIS
LIN {X 93.4823,Y -15.9341,Z 92,A -14.2302,B 24.9249,C -2.0005,E1 25.1576,E2 99.4165} C_DIS
LIN {X 93.8055,Y -13.9147,Z 92,A -12.8468,B 24.9242,C -2.0101,E1 25.1582,E2 98.0187} C_DIS
LIN {X 94.1516,Y -11.3279,Z 92,A -11.4369,B 24.9243,C -2.0088,E1 25.1587,E2 96.6201} C_DIS
LIN {X 94.407,Y -8.9507,Z 92,A -10.0379,B 24.9241,C -2.0117,E1 25.1591,E2 95.2226} C_DIS
LIN {X 94.594,Y -6.6945,Z 92,A -8.4882,B 24.9233,C -2.0231,E1 25.1595,E2 93.6552} C_DIS
LIN {X 94.7676,Y -3.4905,Z 92,A -6.4372,B 24.9225,C -2.0336,E1 25.1597,E2 91.5916} C_DIS
LIN {X 94.8248,Y -1.1637,Z 92,A -4.9404,B 24.9218,C -2.0416,E1 25.1597,E2 90.0848} C_DIS
LIN {X 94.7947,Y 2.6096,Z 92,A -2.9021,B 24.922,C -2.0396,E1 25.1597,E2 88.0632} C_DIS
LIN {X 94.6391,Y 6.027,Z 92,A -0.8198,B 24.9214,C -2.0468,E1 25.1594,E2 85.9764} C_DIS
LIN {X 94.4563,Y 8.4176,Z 92,A 0.5889,B 24.9212,C -2.0499,E1 25.1591,E2 84.5688} C_DIS
LIN {X 94.0824,Y 11.8885,Z 92,A 2.7774,B 24.9205,C -2.0596,E1 25.1584,E2 82.3703} C_DIS
LIN {X 93.6277,Y 15.0648,Z 92,A 4.6092,B 24.9203,C -2.0616,E1 25.1576,E2 80.5446} C_DIS
LIN {X 93.1764,Y 17.6354,Z 92,A 6.0188,B 24.9204,C -2.0601,E1 25.1569,E2 79.1466} C_DIS
LIN {X 92.7155,Y 19.9167,Z 92,A 7.4155,B 24.9201,C -2.0641,E1 25.1561,E2 77.7486} C_DIS
LIN {X 92.2657,Y 21.9117,Z 92,A 8.7994,B 24.9194,C -2.0736,E1 25.1552,E2 76.3505} C_DIS
LIN {X 91.6266,Y 24.4421,Z 92,A 10.3935,B 24.9189,C -2.0791,E1 25.1541,E2 74.7526} C_DIS
LIN {X 90.7485,Y 27.5282,Z 92,A 12.4178,B 24.9182,C -2.0882,E1 25.1525,E2 72.7183} C_DIS
LIN {X 90.0456,Y 29.747,Z 92,A 13.8148,B 24.9179,C -2.092,E1 25.1513,E2 71.3202} C_DIS
LIN {X 89.1916,Y 32.2132,Z 92,A 15.3637,B 24.9176,C -2.0957,E1 25.1499,E2 69.7715} C_DIS
LIN {X 88.052,Y 35.2127,Z 92,A 17.1821,B 24.9176,C -2.0967,E1 25.148,E2 67.9607} C_DIS
LIN {X 87.1613,Y 37.363,Z 92,A 18.5796,B 24.9173,C -2.1004,E1 25.1465,E2 66.5621} C_DIS
LIN {X 86.0989,Y 39.7469,Z 92,A 19.99,B 24.9174,C -2.0986,E1 25.1449,E2 65.1636} C_DIS
LIN {X 85.0976,Y 41.8479,Z 92,A 21.5444,B 24.9166,C -2.1082,E1 25.143,E2 63.595} C_DIS
LIN {X 84.0449,Y 43.9237,Z 92,A 23.0332,B 24.9161,C -2.1152,E1 25.1411,E2 62.0976} C_DIS
LIN {X 82.512,Y 46.7425,Z 92,A 24.9957,B 24.9156,C -2.1213,E1 25.1384,E2 60.1309} C_DIS
LIN {X 81.34,Y 48.7533,Z 92,A 26.3935,B 24.9153,C -2.1247,E1 25.1364,E2 58.7321} C_DIS
LIN {X 80.1191,Y 50.7348,Z 92,A 27.7918,B 24.9151,C -2.1281,E1 25.1343,E2 57.333} C_DIS
LIN {X 78.8498,Y 52.6858,Z 92,A 29.0642,B 24.9151,C -2.1266,E1 25.1324,E2 56.0703} C_DIS
LIN {X 77.1744,Y 55.1077,Z 92,A 30.9334,B 24.9145,C -2.1345,E1 25.1294,E2 54.1917} C_DIS
LIN {X 75.2983,Y 57.6455,Z 92,A 32.7305,B 24.9145,C -2.135,E1 25.1264,E2 52.4019} C_DIS
LIN {X 73.306,Y 60.1607,Z 92,A 34.7853,B 24.9138,C -2.144,E1 25.1228,E2 50.3356} C_DIS
LIN {X 71.6218,Y 62.1544,Z 92,A 36.2281,B 24.9138,C -2.1426,E1 25.1201,E2 48.9025} C_DIS
LIN {X 69.9184,Y 64.0638,Z 92,A 37.8531,B 24.9134,C -2.149,E1 25.1171,E2 47.2695} C_DIS
LIN {X 67.6756,Y 66.4293,Z 92,A 39.5702,B 24.9138,C -2.1439,E1 25.1138,E2 45.5719} C_DIS
LIN {X 66.2283,Y 67.8741,Z 92,A 41.0829,B 24.9128,C -2.1568,E1 25.1108,E2 44.0351} C_DIS
LIN {X 64.5306,Y 69.49,Z 92,A 42.4852,B 24.9126,C -2.1592,E1 25.1079,E2 42.633} C_DIS
LIN {X 62.6054,Y 71.2278,Z 92,A 43.9268,B 24.9126,C -2.1577,E1 25.1049,E2 41.2007} C_DIS
LIN {X 60.7187,Y 72.8424,Z 92,A 45.3587,B 24.9126,C -2.158,E1 25.1019,E2 39.7735} C_DIS
LIN {X 58.1198,Y 74.9328,Z 92,A 47.2713,B 24.9126,C -2.158,E1 25.0977,E2 37.8682} C_DIS
LIN {X 56.4913,Y 76.1697,Z 92,A 48.6589,B 24.912,C -2.1657,E1 25.0946,E2 36.4673} C_DIS
LIN {X 54.3495,Y 77.7107,Z 92,A 50.0743,B 24.9123,C -2.1619,E1 25.0914,E2 35.0659} C_DIS
LIN {X 52.6858,Y 78.8498,Z 92,A 51.5877,B 24.9113,C -2.1746,E1 25.0878,E2 33.5274} C_DIS
LIN {X 50.4953,Y 80.2687,Z 92,A 53.1455,B 24.9112,C -2.1764,E1 25.0842,E2 31.9704} C_DIS
LIN {X 47.7349,Y 81.9417,Z 92,A 55.0943,B 24.9109,C -2.1792,E1 25.0795,E2 30.021} C_DIS
LIN {X 44.7034,Y 83.6343,Z 92,A 57.0682,B 24.9111,C -2.1776,E1 25.0747,E2 28.0567} C_DIS
LIN {X 42.4615,Y 84.7934,Z 92,A 58.4796,B 24.9112,C -2.1754,E1 25.0712,E2 26.6542} C_DIS
LIN {X 40.2898,Y 85.8462,Z 92,A 60.0431,B 24.9108,C -2.181,E1 25.0672,E2 25.0816} C_DIS
LIN {X 37.363,Y 87.1613,Z 92,A 61.9774,B 24.9106,C -2.183,E1 25.0623,E2 23.1473} C_DIS
LIN {X 35.2127,Y 88.052,Z 92,A 63.3805,B 24.9106,C -2.1843,E1 25.0586,E2 21.7443} C_DIS
LIN {X 32.703,Y 89.013,Z 92,A 64.9688,B 24.9105,C -2.1846,E1 25.0545,E2 20.1587} C_DIS
LIN {X 29.747,Y 90.0456,Z 92,A 67.0157,B 24.9099,C -2.1917,E1 25.0491,E2 18.099} C_DIS
LIN {X 27.2575,Y 90.8288,Z 92,A 68.4463,B 24.9102,C -2.1877,E1 25.0453,E2 16.6804} C_DIS
LIN {X 24.1694,Y 91.7002,Z 92,A 70.5258,B 24.9097,C -2.194,E1 25.0396,E2 14.5894} C_DIS
LIN {X 20.7778,Y 92.5277,Z 92,A 72.6329,B 24.9097,C -2.195,E1 25.0339,E2 12.4828} C_DIS
LIN {X 18.2234,Y 93.0631,Z 92,A 74.1372,B 24.9097,C -2.1932,E1 25.0298,E2 10.9847} C_DIS
LIN {X 15.3434,Y 93.5811,Z 92,A 75.8788,B 24.9098,C -2.1929,E1 25.025,E2 9.2456} C_DIS
LIN {X 12.7625,Y 93.9692,Z 92,A 77.551,B 24.9095,C -2.1966,E1 25.0204,E2 7.5661} C_DIS
LIN {X 10.4526,Y 94.2541,Z 92,A 78.8565,B 24.9098,C -2.1933,E1 25.0168,E2 6.2693} C_DIS
LIN {X 8.1363,Y 94.4822,Z 92,A 80.3626,B 24.9095,C -2.1969,E1 25.0126,E2 4.7555} C_DIS
LIN {X 5.1058,Y 94.6926,Z 92,A 82.1422,B 24.9096,C -2.195,E1 25.0076,E2 2.9812} C_DIS
LIN {X 2.0449,Y 94.8085,Z 92,A 83.7648,B 24.9103,C -2.187,E1 25.0032,E2 1.3781} C_DIS
LIN {X -0.2824,Y 94.8302,Z 92,A 85.1716,B 24.9103,C -2.1867,E1 24.9992,E2 -0.028} C_DIS
LIN {X -2.6096,Y 94.7947,Z 92,A 86.7367,B 24.9099,C -2.1918,E1 24.9948,E2 -1.6054} C_DIS
LIN {X -6.1231,Y 94.6326,Z 92,A 89.0006,B 24.9096,C -2.1958,E1 24.9885,E2 -3.8794} C_DIS
LIN {X -9.5761,Y 94.3458,Z 92,A 90.8013,B 24.9105,C -2.1848,E1 24.9835,E2 -5.6548} C_DIS
LIN {X -11.8885,Y 94.0824,Z 92,A 92.3671,B 24.9101,C -2.1894,E1 24.9792,E2 -7.2327} C_DIS
LIN {X -15.0648,Y 93.6277,Z 92,A 94.4357,B 24.9098,C -2.1925,E1 24.9734,E2 -9.3104} C_DIS
LIN {X -17.358,Y 93.2298,Z 92,A 95.717,B 24.9103,C -2.1872,E1 24.9699,E2 -10.5804} C_DIS
LIN {X -19.9167,Y 92.7155,Z 92,A 97.2969,B 24.9103,C -2.186,E1 24.9656,E2 -12.1594} C_DIS
LIN {X -23.3158,Y 91.9196,Z 92,A 99.4109,B 24.9105,C -2.1842,E1 24.9599,E2 -14.2719} C_DIS
LIN {X -26.6833,Y 90.9991,Z 92,A 101.6181,B 24.9105,C -2.1853,E1 24.9539,E2 -16.4851} C_DIS
LIN {X -29.747,Y 90.0456,Z 92,A 103.4686,B 24.9109,C -2.18,E1 24.949,E2 -18.3264} C_DIS
LIN {X -31.9479,Y 89.2884,Z 92,A 105.0061,B 24.9106,C -2.1827,E1 24.945,E2 -19.8733} C_DIS
LIN {X -34.3924,Y 88.3742,Z 92,A 106.4698,B 24.9111,C -2.1768,E1 24.9412,E2 -21.3262} C_DIS
LIN {X -36.5509,Y 87.5036,Z 92,A 107.8708,B 24.9113,C -2.1747,E1 24.9376,E2 -22.7252} C_DIS
LIN {X -39.4908,Y 86.2181,Z 92,A 109.9434,B 24.9112,C -2.1762,E1 24.9323,E2 -24.8065} C_DIS
LIN {X -41.8479,Y 85.0976,Z 92,A 111.3981,B 24.9117,C -2.1697,E1 24.9286,E2 -26.2495} C_DIS
LIN {X -44.7034,Y 83.6343,Z 92,A 113.344,B 24.9119,C -2.1667,E1 24.9238,E2 -28.1935} C_DIS
LIN {X -46.9345,Y 82.4016,Z 92,A 114.9162,B 24.9121,C -2.1651,E1 24.92,E2 -29.7665} C_DIS
LIN {X -49.9874,Y 80.586,Z 92,A 116.8864,B 24.9129,C -2.1555,E1 24.9153,E2 -31.7198} C_DIS
LIN {X -51.95,Y 79.335,Z 92,A 118.457,B 24.9126,C -2.1582,E1 24.9116,E2 -33.3018} C_DIS
LIN {X -53.8813,Y 78.0361,Z 92,A 119.8693,B 24.9128,C -2.1556,E1 24.9083,E2 -34.7128} C_DIS
LIN {X -55.7802,Y 76.6903,Z 92,A 121.2818,B 24.9131,C -2.1529,E1 24.9051,E2 -36.1239} C_DIS
LIN {X -58.3436,Y 74.7604,Z 92,A 123.2295,B 24.9134,C -2.1491,E1 24.9008,E2 -38.0696} C_DIS
LIN {X -60.1607,Y 73.306,Z 92,A 124.7699,B 24.9133,C -2.1504,E1 24.8975,E2 -39.6189} C_DIS
LIN {X -62.157,Y 71.6195,Z 92,A 126.3624,B 24.9135,C -2.1474,E1 24.8941,E2 -41.2103} C_DIS
LIN {X -64.5427,Y 69.479,Z 92,A 128.3032,B 24.9139,C -2.143,E1 24.8901,E2 -43.1485} C_DIS
LIN {X -67.0563,Y 67.0563,Z 92,A 130.296,B 24.9146,C -2.1342,E1 24.8862,E2 -45.1287} C_DIS
LIN {X -68.6817,Y 65.3904,Z 92,A 131.8374,B 24.9145,C -2.1351,E1 24.8832,E2 -46.679} C_DIS
LIN {X -70.2658,Y 63.6852,Z 92,A 133.2209,B 24.9148,C -2.1309,E1 24.8806,E2 -48.0585} C_DIS
LIN {X -71.9907,Y 61.7266,Z 92,A 134.7097,B 24.9154,C -2.1241,E1 24.8778,E2 -49.5378} C_DIS
LIN {X -74.0388,Y 59.2566,Z 92,A 136.6596,B 24.9158,C -2.1194,E1 24.8744,E2 -51.4854} C_DIS
LIN {X -75.6404,Y 57.1959,Z 92,A 138.2748,B 24.916,C -2.1164,E1 24.8717,E2 -53.1014} C_DIS
LIN {X -77.0212,Y 55.3224,Z 92,A 139.6605,B 24.9164,C -2.1119,E1 24.8694,E2 -54.4831} C_DIS
LIN {X -78.8498,Y 52.6858,Z 92,A 141.7387,B 24.9164,C -2.111,E1 24.8661,E2 -56.5694} C_DIS
LIN {X -80.1191,Y 50.7348,Z 92,A 143.1535,B 24.9167,C -2.1073,E1 24.864,E2 -57.9827} C_DIS
LIN {X -81.34,Y 48.7533,Z 92,A 144.5687,B 24.917,C -2.1036,E1 24.8619,E2 -59.3962} C_DIS
LIN {X -82.6497,Y 46.4959,Z 92,A 146.0281,B 24.9177,C -2.0954,E1 24.8599,E2 -60.8435} C_DIS
LIN {X -84.1765,Y 43.6738,Z 92,A 148.1067,B 24.9177,C -2.0941,E1 24.8572,E2 -62.9302} C_DIS
LIN {X -85.223,Y 41.5948,Z 92,A 149.3943,B 24.9184,C -2.0862,E1 24.8556,E2 -64.2059} C_DIS
LIN {X -86.4328,Y 39.0144,Z 92,A 151.0341,B 24.919,C -2.0785,E1 24.8537,E2 -65.8362} C_DIS
LIN {X -87.6132,Y 36.2906,Z 92,A 153.0612,B 24.9188,C -2.0804,E1 24.8515,E2 -67.8791} C_DIS
LIN {X -88.5775,Y 33.8654,Z 92,A 154.5545,B 24.9194,C -2.0729,E1 24.85,E2 -69.3629} C_DIS
LIN {X -89.764,Y 30.5821,Z 92,A 156.4861,B 24.9204,C -2.0608,E1 24.8482,E2 -71.2767} C_DIS
LIN {X -90.4875,Y 28.37,Z 92,A 157.9018,B 24.9207,C -2.0568,E1 24.847,E2 -72.6907} C_DIS
LIN {X -91.1564,Y 26.1408,Z 92,A 159.3179,B 24.921,C -2.0527,E1 24.8459,E2 -74.1052} C_DIS
LIN {X -91.7002,Y 24.1694,Z 92,A 160.9334,B 24.9204,C -2.0607,E1 24.8447,E2 -75.7493} C_DIS
LIN {X -92.5277,Y 20.7778,Z 92,A 162.9728,B 24.9211,C -2.0518,E1 24.8434,E2 -77.7795} C_DIS
LIN {X -93.0097,Y 18.5008,Z 92,A 164.3889,B 24.9214,C -2.0477,E1 24.8426,E2 -79.194} C_DIS
LIN {X -93.6277,Y 15.0648,Z 92,A 166.5959,B 24.9217,C -2.044,E1 24.8416,E2 -81.4054} C_DIS
LIN {X -94.1187,Y 11.6084,Z 92,A 168.5099,B 24.9226,C -2.0311,E1 24.8409,E2 -83.3001} C_DIS
LIN {X -94.4007,Y 9.0198,Z 92,A 169.9521,B 24.9233,C -2.022,E1 24.8405,E2 -84.7291} C_DIS
LIN {X -94.594,Y 6.6945,Z 92,A 171.5138,B 24.9233,C -2.0222,E1 24.8401,E2 -86.3008} C_DIS
LIN {X -94.7676,Y 3.4905,Z 92,A 173.5941,B 24.9235,C -2.0204,E1 24.8398,E2 -88.3893} C_DIS
LIN {X -94.8282,Y 0.7036,Z 92,A 175.3286,B 24.9237,C -2.0166,E1 24.8398,E2 -90.1252} C_DIS
LIN {X -94.7947,Y -2.6096,Z 92,A 177.1791,B 24.9246,C -2.0054,E1 24.8398,E2 -91.9601} C_DIS
LIN {X -94.6534,Y -5.8152,Z 92,A 179.3202,B 24.9246,C -2.0056,E1 24.8402,E2 -94.1146} C_DIS
LIN {X -94.4563,Y -8.4176,Z 92,A -179.2809,B 24.9254,C -1.995,E1 24.8405,E2 -95.4966} C_DIS
LIN {X -94.0824,Y -11.8885,Z 92,A -177.1568,B 24.9258,C -1.9888,E1 24.8412,E2 -97.6186} C_DIS
LIN {X -93.6277,Y -15.0648,Z 92,A -175.077,B 24.926,C -1.9872,E1 24.8421,E2 -99.7069} C_DIS
LIN {X -93.2298,Y -17.358,Z 92,A -173.789,B 24.9266,C -1.9791,E1 24.8427,E2 -100.9832} C_DIS
LIN {X -92.7155,Y -19.9167,Z 92,A -172.2012,B 24.9269,C -1.9746,E1 24.8436,E2 -102.5695} C_DIS
LIN {X -92.2377,Y -22.0265,Z 92,A -170.7574,B 24.9269,C -1.9749,E1 24.8445,E2 -104.0225} C_DIS
LIN {X -91.3967,Y -25.2929,Z 92,A -168.7059,B 24.9273,C -1.9691,E1 24.846,E2 -106.0722} C_DIS
LIN {X -90.7485,Y -27.5282,Z 92,A -167.2131,B 24.9274,C -1.9676,E1 24.8472,E2 -107.5701} C_DIS
LIN {X -89.7218,Y -30.7073,Z 92,A -165.3766,B 24.9283,C -1.9558,E1 24.8488,E2 -109.389} C_DIS
LIN {X -88.7237,Y -33.4793,Z 92,A -163.669,B 24.9288,C -1.9483,E1 24.8504,E2 -111.0883} C_DIS
LIN {X -87.9455,Y -35.4743,Z 92,A -162.2925,B 24.9289,C -1.9472,E1 24.8519,E2 -112.4698} C_DIS
LIN {X -87.0484,Y -37.6219,Z 92,A -160.7543,B 24.9289,C -1.9474,E1 24.8536,E2 -114.017} C_DIS
LIN {X -85.727,Y -40.5459,Z 92,A -158.9265,B 24.9296,C -1.9384,E1 24.8557,E2 -115.8332} C_DIS
LIN {X -84.7061,Y -42.6375,Z 92,A -157.3842,B 24.9296,C -1.9388,E1 24.8576,E2 -117.3849} C_DIS
LIN {X -83.6343,Y -44.7034,Z 92,A -155.8834,B 24.9296,C -1.938,E1 24.8596,E2 -118.8918} C_DIS
LIN {X -81.9322,Y -47.7515,Z 92,A -153.9751,B 24.9305,C -1.9259,E1 24.8622,E2 -120.7812} C_DIS
LIN {X -80.586,Y -49.9874,Z 92,A -152.5476,B 24.9311,C -1.917,E1 24.8643,E2 -122.1947} C_DIS
LIN {X -79.4904,Y -51.7142,Z 92,A -150.9294,B 24.9304,C -1.9262,E1 24.8667,E2 -123.843} C_DIS
LIN {X -77.5331,Y -54.605,Z 92,A -148.898,B 24.931,C -1.9183,E1 24.87,E2 -125.8658} C_DIS
LIN {X -75.4707,Y -57.4218,Z 92,A -146.7773,B 24.9314,C -1.9136,E1 24.8735,E2 -127.9853} C_DIS
LIN {X -73.7473,Y -59.6163,Z 92,A -145.1062,B 24.9317,C -1.9091,E1 24.8764,E2 -129.6536} C_DIS
LIN {X -71.8075,Y -61.9416,Z 92,A -143.2436,B 24.9319,C -1.906,E1 24.8798,E2 -131.5172} C_DIS
LIN {X -70.0748,Y -63.8933,Z 92,A -141.7863,B 24.9324,C -1.8985,E1 24.8825,E2 -132.9634} C_DIS
LIN {X -68.4857,Y -65.5938,Z 92,A -140.3734,B 24.9326,C -1.8957,E1 24.8852,E2 -134.3756} C_DIS
LIN {X -66.2283,Y -67.8741,Z 92,A -138.4256,B 24.9329,C -1.8919,E1 24.889,E2 -136.3226} C_DIS
LIN {X -64.5427,Y -69.479,Z 92,A -137.0131,B 24.9331,C -1.8892,E1 24.8919,E2 -137.7346} C_DIS
LIN {X -62.6054,Y -71.2278,Z 92,A -135.5877,B 24.9337,C -1.8812,E1 24.8949,E2 -139.1464} C_DIS
LIN {X -60.8385,Y -72.7428,Z 92,A -134.0172,B 24.9335,C -1.8839,E1 24.8982,E2 -140.7295} C_DIS
LIN {X -58.1198,Y -74.9328,Z 92,A -132.0576,B 24.9341,C -1.8751,E1 24.9025,E2 -142.6754} C_DIS
LIN {X -56.2377,Y -76.3554,Z 92,A -130.4819,B 24.9339,C -1.8776,E1 24.906,E2 -144.2627} C_DIS
LIN {X -53.6494,Y -78.1974,Z 92,A -128.4149,B 24.9338,C -1.8794,E1 24.9108,E2 -146.341} C_DIS
LIN {X -51.4765,Y -79.643,Z 92,A -126.8532,B 24.934,C -1.8764,E1 24.9144,E2 -147.9008} C_DIS
LIN {X -48.7533,Y -81.34,Z 92,A -124.8876,B 24.9341,C -1.8744,E1 24.9191,E2 -149.8677} C_DIS
LIN {X -46.7425,Y -82.512,Z 92,A -123.477,B 24.9343,C -1.8726,E1 24.9225,E2 -151.2781} C_DIS
LIN {X -44.2021,Y -83.8983,Z 92,A -121.7372,B 24.9344,C -1.8701,E1 24.9268,E2 -153.0168} C_DIS
LIN {X -41.5948,Y -85.223,Z 92,A -119.9516,B 24.9346,C -1.8685,E1 24.9313,E2 -154.8034} C_DIS
LIN {X -39.4908,Y -86.2181,Z 92,A -118.6689,B 24.935,C -1.8627,E1 24.9345,E2 -156.0754} C_DIS
LIN {X -37.363,Y -87.1613,Z 92,A -117.2592,B 24.935,C -1.8613,E1 24.9381,E2 -157.4851} C_DIS
LIN {X -35.2127,Y -88.052,Z 92,A -115.85,B 24.9351,C -1.86,E1 24.9418,E2 -158.8944} C_DIS
LIN {X -32.7759,Y -88.9864,Z 92,A -114.27,B 24.9352,C -1.8587,E1 24.9459,E2 -160.4746} C_DIS
LIN {X -30.5821,Y -89.764,Z 92,A -112.7382,B 24.935,C -1.8618,E1 24.95,E2 -162.0168} C_DIS
LIN {X -27.4083,Y -90.784,Z 92,A -110.7745,B 24.9352,C -1.8586,E1 24.9552,E2 -163.9763} C_DIS
LIN {X -25.2929,Y -91.3967,Z 92,A -109.5108,B 24.9355,C -1.8554,E1 24.9586,E2 -165.2343} C_DIS
LIN {X -22.7221,Y -92.068,Z 92,A -108.0876,B 24.936,C -1.8482,E1 24.9624,E2 -166.6425} C_DIS
LIN {X -20.7778,Y -92.5277,Z 92,A -106.5683,B 24.9353,C -1.8584,E1 24.9666,E2 -168.1881} C_DIS
LIN {X -17.358,Y -93.2298,Z 92,A -104.4571,B 24.9353,C -1.8577,E1 24.9724,E2 -170.2998} C_DIS
LIN {X -15.0648,Y -93.6277,Z 92,A -103.1769,B 24.9356,C -1.8528,E1 24.9759,E2 -171.5698} C_DIS
LIN {X -12.4122,Y -94.0146,Z 92,A -101.5859,B 24.9357,C -1.8515,E1 24.9803,E2 -173.1589} C_DIS
LIN {X -8.8513,Y -94.4162,Z 92,A -99.2816,B 24.9354,C -1.8562,E1 24.9867,E2 -175.4756} C_DIS
LIN {X -5.5331,Y -94.669,Z 92,A -97.5374,B 24.9361,C -1.8468,E1 24.9915,E2 -177.1983} C_DIS
LIN {X -3.4905,Y -94.7676,Z 92,A -96.018,B 24.9354,C -1.8569,E1 24.9958,E2 -178.742} C_DIS
LIN {X -1.1637,Y -94.8248,Z 92,A -94.6122,B 24.9354,C -1.8571,E1 24.9997,E2 -180.1484} C_DIS
LIN {X -1.1637,Y -94.8248,Z 92,A -94.6122,B 24.9354,C -1.8571,E1 24.9997,E2 -180.1484} C_DIS
Enddeposition()
LIN {X 0.6282,Y -93.8707,Z 92,A -93.7079,B 24.9346,C -1.8677,E1 25.0023,E2 -181.0776} C_DIS
Startdeposition()
$VEL.CP = VEL_PRINT
LIN {X -3.3807,Y -93.8145,Z 92,A -96.9451,B 24.9366,C -1.8397,E1 24.9931,E2 -177.774} C_DIS
LIN {X -6.4122,Y -93.6548,Z 92,A -98.7086,B 24.9363,C -1.8428,E1 24.9882,E2 -176.0171} C_DIS
LIN {X -9.7399,Y -93.3674,Z 92,A -100.9549,B 24.9368,C -1.8358,E1 24.9819,E2 -173.7531} C_DIS
LIN {X -13.1585,Y -92.9473,Z 92,A -102.9438,B 24.9365,C -1.8401,E1 24.9764,E2 -171.7729} C_DIS
LIN {X -16.7759,Y -92.363,Z 92,A -105.2153,B 24.9365,C -1.8396,E1 24.9702,E2 -169.4979} C_DIS
LIN {X -22.545,Y -91.1271,Z 92,A -109.2484,B 24.9374,C -1.8268,E1 24.9591,E2 -165.4294} C_DIS
LIN {X -25.7787,Y -90.2654,Z 92,A -110.5946,B 24.9357,C -1.8515,E1 24.9556,E2 -164.1396} C_DIS
LIN {X -28.3079,Y -89.5058,Z 92,A -112.597,B 24.9366,C -1.8395,E1 24.9502,E2 -162.1053} C_DIS
LIN {X -32.0955,Y -88.2169,Z 92,A -114.8566,B 24.936,C -1.8477,E1 24.9443,E2 -159.8607} C_DIS
LIN {X -35.3727,Y -86.9546,Z 92,A -117.0089,B 24.9359,C -1.8495,E1 24.9387,E2 -157.708} C_DIS
LIN {X -38.4684,Y -85.6302,Z 92,A -119.096,B 24.9359,C -1.8506,E1 24.9333,E2 -155.6186} C_DIS
LIN {X -42.1937,Y -83.8591,Z 92,A -121.5542,B 24.9355,C -1.8556,E1 24.9272,E2 -153.1659} C_DIS
LIN {X -46.4052,Y -81.6031,Z 92,A -125.0093,B 24.9364,C -1.8419,E1 24.9186,E2 -149.6684} C_DIS
LIN {X -49.306,Y -79.8844,Z 92,A -126.4119,B 24.9347,C -1.8663,E1 24.9154,E2 -148.3194} C_DIS
LIN {X -51.55,Y -78.4535,Z 92,A -128.2069,B 24.9349,C -1.8633,E1 24.9112,E2 -146.5113} C_DIS
LIN {X -54.1313,Y -76.6966,Z 92,A -130.0427,B 24.9345,C -1.8686,E1 24.907,E2 -144.6821} C_DIS
LIN {X -56.5492,Y -74.9305,Z 92,A -132.0013,B 24.9346,C -1.8676,E1 24.9026,E2 -142.714} C_DIS
LIN {X -59.3174,Y -72.7589,Z 92,A -134.1067,B 24.9342,C -1.8728,E1 24.898,E2 -140.6133} C_DIS
LIN {X -61.9759,Y -70.5082,Z 92,A -136.1196,B 24.9337,C -1.8806,E1 24.8937,E2 -138.611} C_DIS
LIN {X -64.199,Y -68.4897,Z 92,A -138.1122,B 24.9338,C -1.8791,E1 24.8896,E2 -136.6068} C_DIS
LIN {X -67.8058,Y -64.9215,Z 92,A -141.0814,B 24.9331,C -1.8897,E1 24.8838,E2 -133.6503} C_DIS
LIN {X -69.8203,Y -62.7494,Z 92,A -143.0551,B 24.9331,C -1.8885,E1 24.88,E2 -131.6649} C_DIS
LIN {X -72.2022,Y -59.9931,Z 92,A -145.0858,B 24.9323,C -1.8997,E1 24.8764,E2 -129.6516} C_DIS
LIN {X -73.7213,Y -58.1164,Z 92,A -146.6019,B 24.9322,C -1.9018,E1 24.8737,E2 -128.1336} C_DIS
LIN {X -75.3983,Y -55.926,Z 92,A -148.2943,B 24.9319,C -1.9056,E1 24.8709,E2 -126.4421} C_DIS
LIN {X -77.2231,Y -53.376,Z 92,A -150.2428,B 24.9317,C -1.9093,E1 24.8678,E2 -124.4927} C_DIS
LIN {X -79.2088,Y -50.3831,Z 92,A -152.4567,B 24.9313,C -1.9142,E1 24.8644,E2 -122.2794} C_DIS
LIN {X -80.9264,Y -47.5742,Z 92,A -154.646,B 24.9313,C -1.9139,E1 24.8612,E2 -120.078} C_DIS
LIN {X -82.4446,Y -44.8916,Z 92,A -156.4376,B 24.9308,C -1.9217,E1 24.8588,E2 -118.2958} C_DIS
LIN {X -83.7179,Y -42.4704,Z 92,A -158.1915,B 24.9306,C -1.9237,E1 24.8565,E2 -116.5372} C_DIS
LIN {X -85.2089,Y -39.3934,Z 92,A -160.1665,B 24.9299,C -1.933,E1 24.8542,E2 -114.5738} C_DIS
LIN {X -86.9624,Y -35.3535,Z 92,A -162.726,B 24.9291,C -1.9447,E1 24.8514,E2 -112.028} C_DIS
LIN {X -87.8838,Y -32.9977,Z 92,A -164.6196,B 24.9296,C -1.9384,E1 24.8495,E2 -110.1085} C_DIS
LIN {X -88.9317,Y -30.058,Z 92,A -166.3028,B 24.9286,C -1.9509,E1 24.848,E2 -108.4456} C_DIS
LIN {X -89.8059,Y -27.3398,Z 92,A -168.1983,B 24.9286,C -1.9513,E1 24.8464,E2 -106.5403} C_DIS
LIN {X -90.7989,Y -23.8355,Z 92,A -170.2365,B 24.9277,C -1.9638,E1 24.8449,E2 -104.52} C_DIS
LIN {X -91.6033,Y -20.5296,Z 92,A -172.5539,B 24.9277,C -1.9627,E1 24.8434,E2 -102.1865} C_DIS
LIN {X -92.2612,Y -17.3316,Z 92,A -174.3827,B 24.9269,C -1.9739,E1 24.8424,E2 -100.3736} C_DIS
LIN {X -92.7524,Y -14.4686,Z 92,A -176.3236,B 24.9269,C -1.9743,E1 24.8415,E2 -98.4222} C_DIS
LIN {X -93.2634,Y -10.6928,Z 92,A -178.6911,B 24.9265,C -1.9804,E1 24.8407,E2 -96.0549} C_DIS
LIN {X -93.5927,Y -7.2652,Z 92,A 178.2991,B 24.928,C -1.9595,E1 24.84,E2 -92.9772} C_DIS
LIN {X -93.8453,Y -2.348,Z 92,A 176.3978,B 24.9248,C -2.0026,E1 24.8398,E2 -91.1673} C_DIS
LIN {X -93.8729,Y 0.5315,Z 92,A 173.942,B 24.926,C -1.9869,E1 24.8398,E2 -88.6593} C_DIS
LIN {X -93.7938,Y 3.8838,Z 92,A 171.7189,B 24.9259,C -1.9882,E1 24.8401,E2 -86.4259} C_DIS
LIN {X -93.5469,Y 7.8389,Z 92,A 170.1098,B 24.9234,C -2.0205,E1 24.8404,E2 -84.8843} C_DIS
LIN {X -93.2827,Y 10.5276,Z 92,A 168.2124,B 24.9236,C -2.0182,E1 24.841,E2 -82.97} C_DIS
LIN {X -92.6016,Y 15.4043,Z 92,A 164.9188,B 24.9236,C -2.0191,E1 24.8424,E2 -79.6588} C_DIS
LIN {X -91.6768,Y 20.1925,Z 92,A 162.2418,B 24.9221,C -2.0377,E1 24.8439,E2 -77.0104} C_DIS
LIN {X -90.9284,Y 23.3316,Z 92,A 160.5338,B 24.921,C -2.0519,E1 24.845,E2 -75.3264} C_DIS
LIN {X -90.275,Y 25.7446,Z 92,A 158.7772,B 24.9212,C -2.0496,E1 24.8463,E2 -73.5541} C_DIS
LIN {X -89.3286,Y 28.8573,Z 92,A 156.7641,B 24.9208,C -2.055,E1 24.848,E2 -71.5423} C_DIS
LIN {X -88.0095,Y 32.664,Z 92,A 154.4029,B 24.92,C -2.0655,E1 24.8502,E2 -69.1929} C_DIS
LIN {X -86.9993,Y 35.263,Z 92,A 152.5475,B 24.92,C -2.066,E1 24.8521,E2 -67.3282} C_DIS
LIN {X -85.4303,Y 38.912,Z 92,A 149.9457,B 24.9198,C -2.0679,E1 24.855,E2 -64.7166} C_DIS
LIN {X -83.165,Y 43.5428,Z 92,A 146.6323,B 24.9195,C -2.0721,E1 24.8592,E2 -61.3954} C_DIS
LIN {X -80.8121,Y 47.7676,Z 92,A 144.0636,B 24.9179,C -2.0924,E1 24.8627,E2 -58.8616} C_DIS
LIN {X -79.1094,Y 50.538,Z 92,A 141.9523,B 24.9178,C -2.094,E1 24.8658,E2 -56.7436} C_DIS
LIN {X -77.2596,Y 53.3235,Z 92,A 139.8543,B 24.9175,C -2.0979,E1 24.8691,E2 -54.6444} C_DIS
LIN {X -75.6205,Y 55.623,Z 92,A 138.2711,B 24.9167,C -2.1069,E1 24.8717,E2 -53.075} C_DIS
LIN {X -73.9934,Y 57.7722,Z 92,A 136.6751,B 24.9163,C -2.1128,E1 24.8744,E2 -51.4855} C_DIS
LIN {X -72.3036,Y 59.8711,Z 92,A 134.9203,B 24.9163,C -2.1137,E1 24.8775,E2 -49.7246} C_DIS
LIN {X -70.2243,Y 62.2979,Z 92,A 133.0231,B 24.9157,C -2.1203,E1 24.881,E2 -47.8346} C_DIS
LIN {X -68.4648,Y 64.2256,Z 92,A 131.2634,B 24.9157,C -2.1191,E1 24.8843,E2 -46.0643} C_DIS
LIN {X -65.8982,Y 66.8564,Z 92,A 129.1539,B 24.915,C -2.1287,E1 24.8885,E2 -43.9686} C_DIS
LIN {X -63.7233,Y 68.9333,Z 92,A 127.2726,B 24.9148,C -2.1315,E1 24.8923,E2 -42.0864} C_DIS
LIN {X -61.3322,Y 71.0705,Z 92,A 125.2285,B 24.9147,C -2.1332,E1 24.8966,E2 -40.0383} C_DIS
LIN {X -59.2287,Y 72.8308,Z 92,A 123.6696,B 24.9141,C -2.1406,E1 24.8999,E2 -38.4909} C_DIS
LIN {X -56.9018,Y 74.6644,Z 92,A 121.6726,B 24.9142,C -2.1384,E1 24.9043,E2 -36.4814} C_DIS
LIN {X -54.5139,Y 76.4236,Z 92,A 119.9376,B 24.9137,C -2.1445,E1 24.9082,E2 -34.7549} C_DIS
LIN {X -52.2203,Y 78.0104,Z 92,A 118.3487,B 24.9132,C -2.1514,E1 24.9119,E2 -33.1771} C_DIS
LIN {X -49.7141,Y 79.6294,Z 92,A 116.3621,B 24.9133,C -2.1496,E1 24.9166,E2 -31.1799} C_DIS
LIN {X -46.5816,Y 81.5017,Z 92,A 114.0946,B 24.9131,C -2.1523,E1 24.9221,E2 -28.912} C_DIS
LIN {X -43.5418,Y 83.1655,Z 92,A 112.1597,B 24.9124,C -2.1616,E1 24.9268,E2 -26.9939} C_DIS
LIN {X -40.8318,Y 84.5289,Z 92,A 109.9057,B 24.9132,C -2.1517,E1 24.9325,E2 -24.7103} C_DIS
LIN {X -37.6657,Y 85.9864,Z 92,A 108.0088,B 24.9123,C -2.1622,E1 24.9373,E2 -22.8339} C_DIS
LIN {X -31.1107,Y 88.569,Z 92,A 103.7584,B 24.9117,C -2.1696,E1 24.9484,E2 -18.592} C_DIS
LIN {X -27.6993,Y 89.6945,Z 92,A 101.5839,B 24.9115,C -2.1727,E1 24.9541,E2 -16.421} C_DIS
LIN {X -24.4262,Y 90.6405,Z 92,A 99.4074,B 24.9115,C -2.1717,E1 24.96,E2 -14.2387} C_DIS
LIN {X -21.0674,Y 91.4795,Z 92,A 97.3753,B 24.9112,C -2.1764,E1 24.9655,E2 -12.2149} C_DIS
LIN {X -17.5029,Y 92.2282,Z 92,A 95.247,B 24.9108,C -2.1813,E1 24.9713,E2 -10.0959} C_DIS
LIN {X -15.1181,Y 92.6494,Z 92,A 93.5432,B 24.9113,C -2.1749,E1 24.976,E2 -8.3753} C_DIS
LIN {X -8.6134,Y 93.4781,Z 92,A 90.0738,B 24.9096,C -2.195,E1 24.9855,E2 -4.9512} C_DIS
LIN {X -4.9029,Y 93.7463,Z 92,A 87.1473,B 24.9114,C -2.174,E1 24.9938,E2 -1.9737} C_DIS
LIN {X -0.0777,Y 93.8747,Z 92,A 84.1894,B 24.9114,C -2.1743,E1 25.002,E2 0.9837} C_DIS
LIN {X 4.1671,Y 93.7816,Z 92,A 81.7242,B 24.911,C -2.1788,E1 25.0089,E2 3.4376} C_DIS
LIN {X 8.707,Y 93.4694,Z 92,A 79.1782,B 24.9103,C -2.1865,E1 25.0159,E2 5.9641} C_DIS
LIN {X 11.53,Y 93.1647,Z 92,A 76.8782,B 24.9119,C -2.1669,E1 25.0224,E2 8.3088} C_DIS
LIN {X 16.3111,Y 92.4466,Z 92,A 73.8237,B 24.9123,C -2.1624,E1 25.0309,E2 11.3708} C_DIS
LIN {X 19.6842,Y 91.7877,Z 92,A 71.679,B 24.9125,C -2.1598,E1 25.0367,E2 13.5189} C_DIS
LIN {X 23.1774,Y 90.968,Z 92,A 70.0524,B 24.911,C -2.1778,E1 25.041,E2 15.1003} C_DIS
LIN {X 26.9728,Y 89.916,Z 92,A 67.6108,B 24.9113,C -2.1749,E1 25.0476,E2 17.5449} C_DIS
LIN {X 30.2661,Y 88.8616,Z 92,A 65.6751,B 24.9109,C -2.1792,E1 25.0527,E2 19.4666} C_DIS
LIN {X 33.0364,Y 87.8691,Z 92,A 63.722,B 24.9115,C -2.1721,E1 25.0578,E2 21.4324} C_DIS
LIN {X 36.2119,Y 86.6089,Z 92,A 61.6973,B 24.9115,C -2.1721,E1 25.0631,E2 23.4527} C_DIS
LIN {X 39.8444,Y 84.999,Z 92,A 58.6314,B 24.9136,C -2.1469,E1 25.071,E2 26.5703} C_DIS
LIN {X 43.3143,Y 83.2853,Z 92,A 56.2579,B 24.9138,C -2.1434,E1 25.0769,E2 28.9455} C_DIS
LIN {X 46.6764,Y 81.4473,Z 92,A 54.9606,B 24.9111,C -2.1769,E1 25.0798,E2 30.1598} C_DIS
LIN {X 50.1332,Y 79.3676,Z 92,A 52.0291,B 24.9128,C -2.1565,E1 25.0869,E2 33.1304} C_DIS
LIN {X 53.1918,Y 77.3511,Z 92,A 49.8309,B 24.913,C -2.1542,E1 25.092,E2 35.3266} C_DIS
LIN {X 57.1232,Y 74.4938,Z 92,A 46.5297,B 24.9143,C -2.1371,E1 25.0994,E2 38.6565} C_DIS
LIN {X 60.1343,Y 72.0849,Z 92,A 44.4917,B 24.9138,C -2.1439,E1 25.1038,E2 40.6705} C_DIS
LIN {X 62.7345,Y 69.8337,Z 92,A 42.5801,B 24.9136,C -2.1465,E1 25.1078,E2 42.5683} C_DIS
LIN {X 65.7265,Y 67.026,Z 92,A 40.0268,B 24.9141,C -2.1396,E1 25.1129,E2 45.1276} C_DIS
LIN {X 68.3057,Y 64.3948,Z 92,A 37.7589,B 24.9146,C -2.134,E1 25.1173,E2 47.3987} C_DIS
LIN {X 71.1449,Y 61.2451,Z 92,A 35.3714,B 24.9145,C -2.1354,E1 25.1217,E2 49.7722} C_DIS
LIN {X 73.5,Y 58.3964,Z 92,A 33.0453,B 24.9151,C -2.1276,E1 25.1259,E2 52.1062} C_DIS
LIN {X 76.1717,Y 54.867,Z 92,A 28.9652,B 24.9196,C -2.071,E1 25.1328,E2 56.3001} C_DIS
LIN {X 79.6155,Y 49.7364,Z 92,A 26.6317,B 24.9162,C -2.1135,E1 25.1361,E2 58.5217} C_DIS
LIN {X 80.9606,Y 47.5163,Z 92,A 25.0569,B 24.9165,C -2.1096,E1 25.1384,E2 60.0976} C_DIS
LIN {X 82.1702,Y 45.3936,Z 92,A 23.1245,B 24.9181,C -2.0894,E1 25.141,E2 62.0677} C_DIS
LIN {X 84.1931,Y 41.5199,Z 92,A 20.7295,B 24.9179,C -2.092,E1 25.144,E2 64.4437} C_DIS
LIN {X 85.6602,Y 38.4018,Z 92,A 18.6934,B 24.9182,C -2.0885,E1 25.1464,E2 66.4769} C_DIS
LIN {X 87.3877,Y 34.2888,Z 92,A 16.1586,B 24.9182,C -2.0877,E1 25.1491,E2 68.9999} C_DIS
LIN {X 88.1011,Y 32.4129,Z 92,A 14.7664,B 24.919,C -2.0778,E1 25.1505,E2 70.4075} C_DIS
LIN {X 89.2726,Y 29.0304,Z 92,A 12.5644,B 24.9196,C -2.0707,E1 25.1524,E2 72.6139} C_DIS
LIN {X 90.3098,Y 25.6217,Z 92,A 10.6096,B 24.9195,C -2.0723,E1 25.154,E2 74.5537} C_DIS
LIN {X 91.549,Y 20.7669,Z 92,A 7.4498,B 24.9205,C -2.0591,E1 25.1561,E2 77.7263} C_DIS
LIN {X 92.6207,Y 15.2896,Z 92,A 4.1643,B 24.921,C -2.0531,E1 25.1578,E2 81.007} C_DIS
LIN {X 93.063,Y 12.3162,Z 92,A 1.738,B 24.9231,C -2.0252,E1 25.1587,E2 83.4847} C_DIS
LIN {X 93.4405,Y 9.0203,Z 92,A 0.227,B 24.9221,C -2.0379,E1 25.1592,E2 84.9568} C_DIS
LIN {X 93.7039,Y 5.6667,Z 92,A -1.8679,B 24.9227,C -2.0298,E1 25.1596,E2 87.0584} C_DIS
LIN {X 93.8409,Y 2.5214,Z 92,A -3.6156,B 24.9227,C -2.0302,E1 25.1597,E2 88.7948} C_DIS
LIN {X 93.8751,Y -0.0204,Z 92,A -5.3214,B 24.9235,C -2.0194,E1 25.1597,E2 90.5159} C_DIS
LIN {X 93.8169,Y -3.2942,Z 92,A -7.155,B 24.9235,C -2.0192,E1 25.1597,E2 92.3391} C_DIS
LIN {X 93.6993,Y -5.7534,Z 92,A -8.6308,B 24.9238,C -2.0153,E1 25.1594,E2 93.8152} C_DIS
LIN {X 93.3744,Y -9.6729,Z 92,A -11.1575,B 24.9248,C -2.0029,E1 25.1588,E2 96.3563} C_DIS
LIN {X 92.8947,Y -13.5285,Z 92,A -13.56,B 24.9254,C -1.9941,E1 25.1579,E2 98.7653} C_DIS
LIN {X 92.338,Y -16.9137,Z 92,A -15.6579,B 24.926,C -1.9873,E1 25.1569,E2 100.8671} C_DIS
LIN {X 90.808,Y -23.8,Z 92,A -19.7096,B 24.9263,C -1.9831,E1 25.1544,E2 104.9051} C_DIS
LIN {X 90.1775,Y -26.0886,Z 92,A -21.1821,B 24.9267,C -1.9776,E1 25.1532,E2 106.3821} C_DIS
LIN {X 89.4226,Y -28.5667,Z 92,A -22.8225,B 24.9272,C -1.9705,E1 25.1519,E2 108.03} C_DIS
LIN {X 88.3384,Y -31.7625,Z 92,A -25.0294,B 24.9281,C -1.9586,E1 25.1498,E2 110.2527} C_DIS
LIN {X 87.3896,Y -34.2841,Z 92,A -26.6272,B 24.9283,C -1.9553,E1 25.1482,E2 111.8494} C_DIS
LIN {X 85.9871,Y -37.6641,Z 92,A -28.7533,B 24.9285,C -1.9525,E1 25.1459,E2 113.9703} C_DIS
LIN {X 84.5931,Y -40.6981,Z 92,A -30.7309,B 24.9288,C -1.9486,E1 25.1436,E2 115.9464} C_DIS
LIN {X 83.1558,Y -43.5602,Z 92,A -32.7618,B 24.9294,C -1.94,E1 25.141,E2 117.9868} C_DIS
LIN {X 81.6249,Y -46.3672,Z 92,A -34.6926,B 24.9298,C -1.9351,E1 25.1383,E2 119.9192} C_DIS
LIN {X 80.0548,Y -49.0273,Z 92,A -36.636,B 24.9303,C -1.9275,E1 25.1355,E2 121.8705} C_DIS
LIN {X 78.3334,Y -51.7322,Z 92,A -38.5694,B 24.9307,C -1.9229,E1 25.1326,E2 123.8052} C_DIS
LIN {X 76.2848,Y -54.7085,Z 92,A -40.5451,B 24.9305,C -1.9253,E1 25.1294,E2 125.7654} C_DIS
LIN {X 73.1153,Y -58.8776,Z 92,A -43.8369,B 24.9314,C -1.9132,E1 25.1238,E2 129.0703} C_DIS
LIN {X 69.4642,Y -63.1447,Z 92,A -47.0663,B 24.9314,C -1.9117,E1 25.1179,E2 132.2887} C_DIS
LIN {X 67.6115,Y -65.1232,Z 92,A -48.9023,B 24.9323,C -1.9009,E1 25.1144,E2 134.1423} C_DIS
LIN {X 64.127,Y -68.5574,Z 92,A -52.3058,B 24.9339,C -1.8784,E1 25.1074,E2 137.5847} C_DIS
LIN {X 61.013,Y -71.3427,Z 92,A -54.4275,B 24.9332,C -1.8883,E1 25.103,E2 139.6747} C_DIS
LIN {X 58.3107,Y -73.5678,Z 92,A -56.5331,B 24.9334,C -1.8847,E1 25.0985,E2 141.7809} C_DIS
LIN {X 55.5465,Y -75.6765,Z 92,A -59.2244,B 24.9352,C -1.8596,E1 25.0923,E2 144.5219} C_DIS
LIN {X 52.6046,Y -77.7502,Z 92,A -60.8762,B 24.9341,C -1.8749,E1 25.0886,E2 146.1318} C_DIS
LIN {X 48.5519,Y -80.3436,Z 92,A -63.6164,B 24.934,C -1.8764,E1 25.0822,E2 148.8596} C_DIS
LIN {X 44.4762,Y -82.6699,Z 92,A -66.4753,B 24.9343,C -1.8715,E1 25.0752,E2 151.7216} C_DIS
LIN {X 41.9021,Y -84.0036,Z 92,A -68.608,B 24.9355,C -1.8555,E1 25.0698,E2 153.8865} C_DIS
LIN {X 38.2216,Y -85.7414,Z 92,A -70.818,B 24.935,C -1.8615,E1 25.0643,E2 156.0767} C_DIS
LIN {X 35.3386,Y -86.9685,Z 92,A -72.8296,B 24.9355,C -1.8552,E1 25.0591,E2 158.0985} C_DIS
LIN {X 31.9964,Y -88.253,Z 92,A -74.8731,B 24.9353,C -1.8573,E1 25.0537,E2 160.1326} C_DIS
LIN {X 29.4759,Y -89.1279,Z 92,A -76.714,B 24.936,C -1.8477,E1 25.0488,E2 161.9928} C_DIS
LIN {X 25.773,Y -90.267,Z 92,A -78.7339,B 24.9353,C -1.8573,E1 25.0435,E2 163.9865} C_DIS
LIN {X 23.1613,Y -90.9722,Z 92,A -80.4671,B 24.9357,C -1.8526,E1 25.0388,E2 165.7279} C_DIS
LIN {X 20.2926,Y -91.655,Z 92,A -82.4367,B 24.9362,C -1.8449,E1 25.0334,E2 167.713} C_DIS
LIN {X 15.3754,Y -92.6064,Z 92,A -85.0465,B 24.9353,C -1.8582,E1 25.0263,E2 170.2884} C_DIS
LIN {X 11.8216,Y -93.127,Z 92,A -87.7717,B 24.9367,C -1.838,E1 25.0187,E2 173.0591} C_DIS
LIN {X 8.0644,Y -93.5276,Z 92,A -90.3211,B 24.9373,C -1.8283,E1 25.0115,E2 175.6299} C_DIS
LIN {X 3.3452,Y -93.8156,Z 92,A -92.7911,B 24.9364,C -1.8416,E1 25.0047,E2 178.0677} C_DIS
LIN {X 0.6282,Y -93.8707,Z 92,A -93.7064,B 24.9347,C -1.867,E1 25.0023,E2 178.9224} C_DIS
Enddeposition()
LIN {X 0.6282,Y -93.8707,Z 92,A -93.7064,B 24.9347,C -1.867,E1 25.0023,E2 178.9224} C_DIS
Startdeposition()
$VEL.CP = VEL_PRINT
LIN {X 2.652,Y -92.8803,Z 92,A -92.3359,B 24.9332,C -1.8882,E1 25.0063,E2 177.502} C_DIS
LIN {X 7.1619,Y -92.6419,Z 92,A -89.386,B 24.9327,C -1.8952,E1 25.0145,E2 174.5368} C_DIS
LIN {X 9.7817,Y -92.4017,Z 92,A -87.136,B 24.931,C -1.9183,E1 25.021,E2 172.2335} C_DIS
LIN {X 14.1667,Y -91.8317,Z 92,A -85.1912,B 24.9329,C -1.8925,E1 25.0261,E2 170.3517} C_DIS
LIN {X 16.6029,Y -91.4227,Z 92,A -83.6158,B 24.9326,C -1.8955,E1 25.0305,E2 168.7708} C_DIS
LIN {X 20.4791,Y -90.6342,Z 92,A -81.224,B 24.9326,C -1.896,E1 25.037,E2 166.3809} C_DIS
LIN {X 23.779,Y -89.825,Z 92,A -79.1905,B 24.9326,C -1.896,E1 25.0425,E2 164.3506} C_DIS
LIN {X 27.447,Y -88.7717,Z 92,A -77.236,B 24.9334,C -1.8844,E1 25.0477,E2 162.4268} C_DIS
LIN {X 31.1567,Y -87.5396,Z 92,A -74.402,B 24.9321,C -1.9025,E1 25.0553,E2 159.5555} C_DIS
LIN {X 34.269,Y -86.3683,Z 92,A -72.4222,B 24.9321,C -1.9028,E1 25.0604,E2 157.5793} C_DIS
LIN {X 36.9396,Y -85.26,Z 92,A -70.7648,B 24.9323,C -1.9009,E1 25.0646,E2 155.9304} C_DIS
LIN {X 41.9882,Y -82.8906,Z 92,A -67.1345,B 24.9314,C -1.9132,E1 25.0739,E2 152.2804} C_DIS
LIN {X 44.2489,Y -81.7055,Z 92,A -65.4204,B 24.9308,C -1.921,E1 25.0781,E2 150.5527} C_DIS
LIN {X 48.4483,Y -79.2878,Z 92,A -62.3362,B 24.9302,C -1.93,E1 25.0855,E2 147.4567} C_DIS
LIN {X 52.0183,Y -76.9925,Z 92,A -60.1406,B 24.9309,C -1.9197,E1 25.0906,E2 145.2927} C_DIS
LIN {X 54.8662,Y -74.9897,Z 92,A -57.8959,B 24.9303,C -1.9277,E1 25.0957,E2 143.037} C_DIS
LIN {X 58.0357,Y -72.5643,Z 92,A -55.0173,B 24.9288,C -1.9484,E1 25.1021,E2 140.12} C_DIS
LIN {X 60.6749,Y -70.3748,Z 92,A -52.9779,B 24.9287,C -1.9504,E1 25.1064,E2 138.084} C_DIS
LIN {X 64.4284,Y -66.9532,Z 92,A -50.0296,B 24.9287,C -1.951,E1 25.1124,E2 135.1463} C_DIS
LIN {X 68.1983,Y -63.1102,Z 92,A -47.141,B 24.9292,C -1.9432,E1 25.1179,E2 132.2887} C_DIS
LIN {X 70.3926,Y -60.6511,Z 92,A -44.7208,B 24.9278,C -1.9628,E1 25.1225,E2 129.833} C_DIS
LIN {X 72.9778,Y -57.5153,Z 92,A -42.0523,B 24.9268,C -1.9755,E1 25.1271,E2 127.1469} C_DIS
LIN {X 75.816,Y -53.7195,Z 92,A -39.4301,B 24.9271,C -1.9722,E1 25.1314,E2 124.5452} C_DIS
LIN {X 77.7729,Y -50.8455,Z 92,A -37.3255,B 24.9267,C -1.9767,E1 25.1347,E2 122.4404} C_DIS
LIN {X 79.556,Y -48.0071,Z 92,A -35.4745,B 24.9269,C -1.9746,E1 25.1374,E2 120.6039} C_DIS
LIN {X 81.3138,Y -44.9658,Z 92,A -32.9091,B 24.9253,C -1.9958,E1 25.1409,E2 118.0016} C_DIS
LIN {X 83.313,Y -41.1425,Z 92,A -30.4411,B 24.9253,C -1.9965,E1 25.1441,E2 115.5452} C_DIS
LIN {X 84.8077,Y -37.9665,Z 92,A -28.3915,B 24.9251,C -1.9987,E1 25.1464,E2 113.5016} C_DIS
LIN {X 85.8909,Y -35.4501,Z 92,A -26.0251,B 24.9228,C -2.0294,E1 25.149,E2 111.0756} C_DIS
LIN {X 87.291,Y -31.8438,Z 92,A -24.7626,B 24.9254,C -1.9944,E1 25.1502,E2 109.9028} C_DIS
LIN {X 88.2314,Y -29.1427,Z 92,A -22.4979,B 24.9236,C -2.0186,E1 25.1523,E2 107.5937} C_DIS
LIN {X 89.1966,Y -26.0363,Z 92,A -20.6914,B 24.9236,C -2.0174,E1 25.1537,E2 105.8002} C_DIS
LIN {X 89.9865,Y -23.1555,Z 92,A -18.2526,B 24.9215,C -2.0459,E1 25.1555,E2 103.3084} C_DIS
LIN {X 90.7572,Y -19.9223,Z 92,A -16.5537,B 24.922,C -2.0391,E1 25.1565,E2 101.6354} C_DIS
LIN {X 91.3255,Y -17.1347,Z 92,A -14.2281,B 24.9199,C -2.0663,E1 25.1577,E2 99.2591} C_DIS
LIN {X 91.9978,Y -13.0443,Z 92,A -12.3271,B 24.9212,C -2.0497,E1 25.1584,E2 97.4086} C_DIS
LIN {X 92.4083,Y -9.7188,Z 92,A -10.3957,B 24.9212,C -2.0512,E1 25.159,E2 95.485} C_DIS
LIN {X 92.6652,Y -6.8706,Z 92,A -8.6715,B 24.9208,C -2.0554,E1 25.1594,E2 93.7612} C_DIS
LIN {X 92.8954,Y -2.0823,Z 92,A -5.3565,B 24.919,C -2.0785,E1 25.1598,E2 90.4115} C_DIS
LIN {X 92.8871,Y 2.4332,Z 92,A -2.8386,B 24.919,C -2.0773,E1 25.1597,E2 87.9113} C_DIS
LIN {X 92.5771,Y 7.972,Z 92,A 0.3481,B 24.919,C -2.0794,E1 25.1591,E2 84.7387} C_DIS
LIN {X 91.9069,Y 13.6803,Z 92,A 3.862,B 24.9181,C -2.0894,E1 25.1579,E2 81.2219} C_DIS
LIN {X 91.2331,Y 17.6147,Z 92,A 6.5966,B 24.9167,C -2.1073,E1 25.1565,E2 78.4609} C_DIS
LIN {X 89.8306,Y 23.7582,Z 92,A 10.2953,B 24.9163,C -2.1122,E1 25.1541,E2 74.7722} C_DIS
LIN {X 89.0659,Y 26.4768,Z 92,A 12.0929,B 24.9157,C -2.1196,E1 25.1527,E2 72.9674} C_DIS
LIN {X 88.0479,Y 29.687,Z 92,A 14.0681,B 24.9156,C -2.122,E1 25.151,E2 70.9977} C_DIS
LIN {X 87.0559,Y 32.4842,Z 92,A 16.0526,B 24.9147,C -2.1331,E1 25.1491,E2 68.9981} C_DIS
LIN {X 84.0158,Y 39.6911,Z 92,A 20.565,B 24.9145,C -2.1352,E1 25.1441,E2 64.5052} C_DIS
LIN {X 81.3869,Y 44.8353,Z 92,A 24.3324,B 24.9131,C -2.1526,E1 25.1392,E2 60.7168} C_DIS
LIN {X 79.6812,Y 47.8011,Z 92,A 26.4076,B 24.9127,C -2.1569,E1 25.1363,E2 58.6421} C_DIS
LIN {X 76.1176,Y 53.2911,Z 92,A 30.443,B 24.9119,C -2.1672,E1 25.1301,E2 54.6025} C_DIS
LIN {X 74.5895,Y 55.4113,Z 92,A 32.2574,B 24.911,C -2.1786,E1 25.127,E2 52.7697} C_DIS
LIN {X 72.0264,Y 58.7027,Z 92,A 34.584,B 24.9112,C -2.1757,E1 25.123,E2 50.4609} C_DIS
LIN {X 70.4823,Y 60.5486,Z 92,A 36.5396,B 24.9095,C -2.1964,E1 25.1194,E2 48.4652} C_DIS
LIN {X 68.1454,Y 63.1676,Z 92,A 38.0039,B 24.9112,C -2.1756,E1 25.1167,E2 47.0566} C_DIS
LIN {X 65.8279,Y 65.5789,Z 92,A 40.0772,B 24.9108,C -2.1805,E1 25.1126,E2 44.9807} C_DIS
LIN {X 63.0399,Y 68.2628,Z 92,A 42.5628,B 24.9101,C -2.189,E1 25.1076,E2 42.4853} C_DIS
LIN {X 60.6277,Y 70.415,Z 92,A 44.7212,B 24.9093,C -2.1988,E1 25.103,E2 40.3121} C_DIS
LIN {X 56.9221,Y 73.4418,Z 92,A 47.7649,B 24.9086,C -2.2076,E1 25.0963,E2 37.2589} C_DIS
LIN {X 52.9161,Y 76.3784,Z 92,A 50.4935,B 24.9091,C -2.2008,E1 25.0902,E2 34.5559} C_DIS
LIN {X 50.588,Y 77.9412,Z 92,A 52.411,B 24.9084,C -2.2103,E1 25.0857,E2 32.6223} C_DIS
LIN {X 46.8464,Y 80.246,Z 92,A 54.8534,B 24.9088,C -2.2048,E1 25.0799,E2 30.2005} C_DIS
LIN {X 41.5303,Y 83.1208,Z 92,A 58.8549,B 24.9076,C -2.2195,E1 25.07,E2 26.1756} C_DIS
LIN {X 38.3347,Y 84.6418,Z 92,A 60.8595,B 24.9079,C -2.2157,E1 25.0649,E2 24.185} C_DIS
LIN {X 35.8909,Y 85.7067,Z 92,A 62.5849,B 24.9075,C -2.2204,E1 25.0605,E2 22.4527} C_DIS
LIN {X 32.5201,Y 87.0423,Z 92,A 64.7981,B 24.9075,C -2.2217,E1 25.0547,E2 20.241} C_DIS
LIN {X 29.6512,Y 88.06,Z 92,A 66.541,B 24.9077,C -2.2187,E1 25.0501,E2 18.5089} C_DIS
LIN {X 27.4473,Y 88.7716,Z 92,A 68.375,B 24.9064,C -2.2339,E1 25.0452,E2 16.6421} C_DIS
LIN {X 22.5955,Y 90.1305,Z 92,A 71.0018,B 24.9076,C -2.2192,E1 25.0382,E2 14.0543} C_DIS
LIN {X 17.9471,Y 91.1682,Z 92,A 74.4021,B 24.9062,C -2.2366,E1 25.0288,E2 10.6171} C_DIS
LIN {X 13.2983,Y 91.9617,Z 92,A 77.8657,B 24.9045,C -2.2566,E1 25.0191,E2 7.1091} C_DIS
Enddeposition()
END
